gfCNCPoint5[7255] = {X 11.7883, Y 22.2776, Z -7.1667, A 0.000, B 0.000, C 0.000 }
gfCNCPoint5[7256] = {X 14.1139, Y 22.1583, Z -7.1667, A 0.000, B 0.000, C 0.000 }
gfCNCPoint5[7257] = {X 16.4362, Y 21.9881, Z -7.1667, A 0.000, B 0.000, C 0.000 }
gfCNCPoint5[7258] = {X 17.0855, Y 21.9056, Z -7.1667, A 0.000, B 0.000, C 0.000 }
gfCNCPoint5[7259] = {X 17.7182, Y 21.7381, Z -7.1667, A 0.000, B 0.000, C 0.000 }
gfCNCPoint5[7260] = {X 17.7565, Y 21.2348, Z -7.1667, A 0.000, B 0.000, C 0.000 }
gfCNCPoint5[7261] = {X 17.6002, Y 20.7548, Z -7.1667, A 0.000, B 0.000, C 0.000 }
gfCNCPoint5[7262] = {X 17.2730, Y 20.3705, Z -7.1667, A 0.000, B 0.000, C 0.000 }
gfCNCPoint5[7263] = {X 16.3395, Y 19.8212, Z -7.1667, A 0.000, B 0.000, C 0.000 }
gfCNCPoint5[7264] = {X 15.3164, Y 19.4659, Z -7.1667, A 0.000, B 0.000, C 0.000 }
gfCNCPoint5[7265] = {X 13.9815, Y 19.2481, Z -7.1667, A 0.000, B 0.000, C 0.000 }
gfCNCPoint5[7266] = {X 12.6299, Y 19.1939, Z -7.1667, A 0.000, B 0.000, C 0.000 }
gfCNCPoint5[7267] = {X 11.2818, Y 19.3044, Z -7.1667, A 0.000, B 0.000, C 0.000 }
gfCNCPoint5[7268] = {X 10.5939, Y 19.4125, Z -7.1667, A 0.000, B 0.000, C 0.000 }
gfCNCPoint5[7269] = {X 9.2120, Y 19.7717, Z -7.1667, A 0.000, B 0.000, C 0.000 }
gfCNCPoint5[7270] = {X 7.9080, Y 20.3531, Z -7.1667, A 0.000, B 0.000, C 0.000 }
gfCNCPoint5[7271] = {X 7.7436, Y 21.1766, Z -7.1667, A 0.000, B 0.000, C 0.000 }
gfCNCPoint5[7272] = {X 7.4229, Y 21.9527, Z -7.1667, A 0.000, B 0.000, C 0.000 }
gfCNCPoint5[7273] = {X 6.9582, Y 22.6522, Z -7.1667, A 0.000, B 0.000, C 0.000 }
gfCNCPoint5[7274] = {X 9.0864, Y 22.4225, Z -7.1667, A 0.000, B 0.000, C 0.000 }
gfCNCPoint5[7275] = {X 11.2233, Y 22.2989, Z -7.1667, A 0.000, B 0.000, C 0.000 }
gfCNCPoint5[7276] = {X 11.5058, Y 22.2886, Z -7.1667, A 0.000, B 0.000, C 0.000 }
gfCNCPoint5[7277] = {X 11.7883, Y 22.2776, Z -7.1667, A 0.000, B 0.000, C 0.000 }
gfCNCPoint5[7278] = {X 15.7558, Y 21.7688, Z -7.1667, A 0.000, B 0.000, C 0.000 }
gfCNCPoint5[7279] = {X 7.7960, Y 22.1697, Z -7.1667, A 0.000, B 0.000, C 0.000 }
gfCNCPoint5[7280] = {X 11.7916, Y 22.3576, Z -7.1667, A 0.000, B 0.000, C 0.000 }
gfCNCPoint5[7281] = {X 14.1184, Y 22.2382, Z -7.1667, A 0.000, B 0.000, C 0.000 }
gfCNCPoint5[7282] = {X 16.4420, Y 22.0679, Z -7.1667, A 0.000, B 0.000, C 0.000 }
gfCNCPoint5[7283] = {X 17.1218, Y 21.9800, Z -7.1667, A 0.000, B 0.000, C 0.000 }
gfCNCPoint5[7284] = {X 17.7833, Y 21.8004, Z -7.1667, A 0.000, B 0.000, C 0.000 }
gfCNCPoint5[7285] = {X 17.8390, Y 21.2530, Z -7.1667, A 0.000, B 0.000, C 0.000 }
gfCNCPoint5[7286] = {X 17.6764, Y 20.7273, Z -7.1667, A 0.000, B 0.000, C 0.000 }
gfCNCPoint5[7287] = {X 17.3214, Y 20.3068, Z -7.1667, A 0.000, B 0.000, C 0.000 }
gfCNCPoint5[7288] = {X 16.3736, Y 19.7488, Z -7.1667, A 0.000, B 0.000, C 0.000 }
gfCNCPoint5[7289] = {X 15.3346, Y 19.3880, Z -7.1667, A 0.000, B 0.000, C 0.000 }
gfCNCPoint5[7290] = {X 13.9897, Y 19.1685, Z -7.1667, A 0.000, B 0.000, C 0.000 }
gfCNCPoint5[7291] = {X 12.6281, Y 19.1140, Z -7.1667, A 0.000, B 0.000, C 0.000 }
gfCNCPoint5[7292] = {X 11.2699, Y 19.2253, Z -7.1667, A 0.000, B 0.000, C 0.000 }
gfCNCPoint5[7293] = {X 10.5808, Y 19.3336, Z -7.1667, A 0.000, B 0.000, C 0.000 }
gfCNCPoint5[7294] = {X 9.6302, Y 19.5537, Z -7.1667, A 0.000, B 0.000, C 0.000 }
gfCNCPoint5[7295] = {X 8.7101, Y 19.8784, Z -7.1667, A 0.000, B 0.000, C 0.000 }
gfCNCPoint5[7296] = {X 7.8318, Y 20.3037, Z -7.1667, A 0.000, B 0.000, C 0.000 }
gfCNCPoint5[7297] = {X 7.8284, Y 20.3451, Z -7.1667, A 0.000, B 0.000, C 0.000 }
gfCNCPoint5[7298] = {X 7.6463, Y 21.2196, Z -7.1667, A 0.000, B 0.000, C 0.000 }
gfCNCPoint5[7299] = {X 7.2851, Y 22.0366, Z -7.1667, A 0.000, B 0.000, C 0.000 }
gfCNCPoint5[7300] = {X 6.7608, Y 22.7597, Z -7.1667, A 0.000, B 0.000, C 0.000 }
gfCNCPoint5[7301] = {X 8.9884, Y 22.5110, Z -7.1667, A 0.000, B 0.000, C 0.000 }
gfCNCPoint5[7302] = {X 11.2260, Y 22.3789, Z -7.1667, A 0.000, B 0.000, C 0.000 }
gfCNCPoint5[7303] = {X 11.5088, Y 22.3686, Z -7.1667, A 0.000, B 0.000, C 0.000 }
gfCNCPoint5[7304] = {X 11.7916, Y 22.3576, Z -7.1667, A 0.000, B 0.000, C 0.000 }
gfCNCPoint5[7305] = {X 15.7591, Y 21.8487, Z -7.1667, A 0.000, B 0.000, C 0.000 }
gfCNCPoint5[7306] = {X 7.7992, Y 22.2496, Z -7.1667, A 0.000, B 0.000, C 0.000 }
gfCNCPoint5[7307] = {X 11.7948, Y 22.4375, Z -7.1667, A 0.000, B 0.000, C 0.000 }
gfCNCPoint5[7308] = {X 14.1229, Y 22.3181, Z -7.1667, A 0.000, B 0.000, C 0.000 }
gfCNCPoint5[7309] = {X 16.4478, Y 22.1477, Z -7.1667, A 0.000, B 0.000, C 0.000 }
gfCNCPoint5[7310] = {X 17.1574, Y 22.0544, Z -7.1667, A 0.000, B 0.000, C 0.000 }
gfCNCPoint5[7311] = {X 17.8470, Y 21.8628, Z -7.1667, A 0.000, B 0.000, C 0.000 }
gfCNCPoint5[7312] = {X 17.9254, Y 21.4214, Z -7.1667, A 0.000, B 0.000, C 0.000 }
gfCNCPoint5[7313] = {X 17.8662, Y 20.9770, Z -7.1667, A 0.000, B 0.000, C 0.000 }
gfCNCPoint5[7314] = {X 17.6750, Y 20.5715, Z -7.1667, A 0.000, B 0.000, C 0.000 }
gfCNCPoint5[7315] = {X 17.3698, Y 20.2431, Z -7.1667, A 0.000, B 0.000, C 0.000 }
gfCNCPoint5[7316] = {X 16.4076, Y 19.6764, Z -7.1667, A 0.000, B 0.000, C 0.000 }
gfCNCPoint5[7317] = {X 15.3528, Y 19.3101, Z -7.1667, A 0.000, B 0.000, C 0.000 }
gfCNCPoint5[7318] = {X 13.9979, Y 19.0889, Z -7.1667, A 0.000, B 0.000, C 0.000 }
gfCNCPoint5[7319] = {X 12.6262, Y 19.0340, Z -7.1667, A 0.000, B 0.000, C 0.000 }
gfCNCPoint5[7320] = {X 11.2580, Y 19.1461, Z -7.1667, A 0.000, B 0.000, C 0.000 }
gfCNCPoint5[7321] = {X 10.5678, Y 19.2546, Z -7.1667, A 0.000, B 0.000, C 0.000 }
gfCNCPoint5[7322] = {X 9.5945, Y 19.4808, Z -7.1667, A 0.000, B 0.000, C 0.000 }
gfCNCPoint5[7323] = {X 8.6531, Y 19.8156, Z -7.1667, A 0.000, B 0.000, C 0.000 }
gfCNCPoint5[7324] = {X 7.7555, Y 20.2547, Z -7.1667, A 0.000, B 0.000, C 0.000 }
gfCNCPoint5[7325] = {X 7.7492, Y 20.3327, Z -7.1667, A 0.000, B 0.000, C 0.000 }
gfCNCPoint5[7326] = {X 7.5473, Y 21.2643, Z -7.1667, A 0.000, B 0.000, C 0.000 }
gfCNCPoint5[7327] = {X 7.1386, Y 22.1254, Z -7.1667, A 0.000, B 0.000, C 0.000 }
gfCNCPoint5[7328] = {X 6.5446, Y 22.8710, Z -7.1667, A 0.000, B 0.000, C 0.000 }
gfCNCPoint5[7329] = {X 8.8810, Y 22.6006, Z -7.1667, A 0.000, B 0.000, C 0.000 }
gfCNCPoint5[7330] = {X 11.2288, Y 22.4588, Z -7.1667, A 0.000, B 0.000, C 0.000 }
gfCNCPoint5[7331] = {X 11.5118, Y 22.4485, Z -7.1667, A 0.000, B 0.000, C 0.000 }
gfCNCPoint5[7332] = {X 11.7948, Y 22.4375, Z -7.1667, A 0.000, B 0.000, C 0.000 }
gfCNCPoint5[7333] = {X 15.7623, Y 21.9287, Z -7.1667, A 0.000, B 0.000, C 0.000 }
gfCNCPoint5[7334] = {X 7.8024, Y 22.3296, Z -7.1667, A 0.000, B 0.000, C 0.000 }
gfCNCPoint5[7335] = {X 11.7980, Y 22.5174, Z -7.1667, A 0.000, B 0.000, C 0.000 }
gfCNCPoint5[7336] = {X 14.1274, Y 22.3980, Z -7.1667, A 0.000, B 0.000, C 0.000 }
gfCNCPoint5[7337] = {X 16.4536, Y 22.2275, Z -7.1667, A 0.000, B 0.000, C 0.000 }
gfCNCPoint5[7338] = {X 17.1925, Y 22.1289, Z -7.1667, A 0.000, B 0.000, C 0.000 }
gfCNCPoint5[7339] = {X 17.9096, Y 21.9253, Z -7.1667, A 0.000, B 0.000, C 0.000 }
gfCNCPoint5[7340] = {X 18.0045, Y 21.4519, Z -7.1667, A 0.000, B 0.000, C 0.000 }
gfCNCPoint5[7341] = {X 17.9481, Y 20.9724, Z -7.1667, A 0.000, B 0.000, C 0.000 }
gfCNCPoint5[7342] = {X 17.7461, Y 20.5338, Z -7.1667, A 0.000, B 0.000, C 0.000 }
gfCNCPoint5[7343] = {X 17.4182, Y 20.1794, Z -7.1667, A 0.000, B 0.000, C 0.000 }
gfCNCPoint5[7344] = {X 16.4416, Y 19.6040, Z -7.1667, A 0.000, B 0.000, C 0.000 }
gfCNCPoint5[7345] = {X 15.3709, Y 19.2322, Z -7.1667, A 0.000, B 0.000, C 0.000 }
gfCNCPoint5[7346] = {X 14.0061, Y 19.0093, Z -7.1667, A 0.000, B 0.000, C 0.000 }
gfCNCPoint5[7347] = {X 12.6243, Y 18.9540, Z -7.1667, A 0.000, B 0.000, C 0.000 }
gfCNCPoint5[7348] = {X 11.2461, Y 19.0670, Z -7.1667, A 0.000, B 0.000, C 0.000 }
gfCNCPoint5[7349] = {X 10.5547, Y 19.1757, Z -7.1667, A 0.000, B 0.000, C 0.000 }
gfCNCPoint5[7350] = {X 9.5588, Y 19.4079, Z -7.1667, A 0.000, B 0.000, C 0.000 }
gfCNCPoint5[7351] = {X 8.5961, Y 19.7528, Z -7.1667, A 0.000, B 0.000, C 0.000 }
gfCNCPoint5[7352] = {X 7.6793, Y 20.2059, Z -7.1667, A 0.000, B 0.000, C 0.000 }
gfCNCPoint5[7353] = {X 7.6695, Y 20.3255, Z -7.1667, A 0.000, B 0.000, C 0.000 }
gfCNCPoint5[7354] = {X 7.5231, Y 21.0760, Z -7.1667, A 0.000, B 0.000, C 0.000 }
gfCNCPoint5[7355] = {X 7.2392, Y 21.7861, Z -7.1667, A 0.000, B 0.000, C 0.000 }
gfCNCPoint5[7356] = {X 6.8279, Y 22.4307, Z -7.1667, A 0.000, B 0.000, C 0.000 }
gfCNCPoint5[7357] = {X 6.3034, Y 22.9872, Z -7.1667, A 0.000, B 0.000, C 0.000 }
gfCNCPoint5[7358] = {X 8.7610, Y 22.6917, Z -7.1667, A 0.000, B 0.000, C 0.000 }
gfCNCPoint5[7359] = {X 11.2315, Y 22.5388, Z -7.1667, A 0.000, B 0.000, C 0.000 }
gfCNCPoint5[7360] = {X 11.5147, Y 22.5285, Z -7.1667, A 0.000, B 0.000, C 0.000 }
gfCNCPoint5[7361] = {X 11.7980, Y 22.5174, Z -7.1667, A 0.000, B 0.000, C 0.000 }
gfCNCPoint5[7362] = {X 15.7655, Y 22.0086, Z -7.1667, A 0.000, B 0.000, C 0.000 }
gfCNCPoint5[7363] = {X 11.7262, Y 22.6004, Z -7.1667, A 0.000, B 0.000, C 0.000 }
gfCNCPoint5[7364] = {X 11.8012, Y 22.5974, Z -7.1667, A 0.000, B 0.000, C 0.000 }
gfCNCPoint5[7365] = {X 14.1319, Y 22.4778, Z -7.1667, A 0.000, B 0.000, C 0.000 }
gfCNCPoint5[7366] = {X 16.4593, Y 22.3073, Z -7.1667, A 0.000, B 0.000, C 0.000 }
gfCNCPoint5[7367] = {X 17.2271, Y 22.2034, Z -7.1667, A 0.000, B 0.000, C 0.000 }
gfCNCPoint5[7368] = {X 17.9713, Y 21.9879, Z -7.1667, A 0.000, B 0.000, C 0.000 }
gfCNCPoint5[7369] = {X 18.0831, Y 21.4827, Z -7.1667, A 0.000, B 0.000, C 0.000 }
gfCNCPoint5[7370] = {X 18.0299, Y 20.9679, Z -7.1667, A 0.000, B 0.000, C 0.000 }
gfCNCPoint5[7371] = {X 17.8171, Y 20.4962, Z -7.1667, A 0.000, B 0.000, C 0.000 }
gfCNCPoint5[7372] = {X 17.4665, Y 20.1156, Z -7.1667, A 0.000, B 0.000, C 0.000 }
gfCNCPoint5[7373] = {X 16.4756, Y 19.5316, Z -7.1667, A 0.000, B 0.000, C 0.000 }
gfCNCPoint5[7374] = {X 15.3891, Y 19.1542, Z -7.1667, A 0.000, B 0.000, C 0.000 }
gfCNCPoint5[7375] = {X 14.0143, Y 18.9297, Z -7.1667, A 0.000, B 0.000, C 0.000 }
gfCNCPoint5[7376] = {X 12.6225, Y 18.8740, Z -7.1667, A 0.000, B 0.000, C 0.000 }
gfCNCPoint5[7377] = {X 11.2342, Y 18.9879, Z -7.1667, A 0.000, B 0.000, C 0.000 }
gfCNCPoint5[7378] = {X 10.5417, Y 19.0968, Z -7.1667, A 0.000, B 0.000, C 0.000 }
gfCNCPoint5[7379] = {X 9.5230, Y 19.3351, Z -7.1667, A 0.000, B 0.000, C 0.000 }
gfCNCPoint5[7380] = {X 8.5390, Y 19.6902, Z -7.1667, A 0.000, B 0.000, C 0.000 }
gfCNCPoint5[7381] = {X 7.6029, Y 20.1573, Z -7.1667, A 0.000, B 0.000, C 0.000 }
gfCNCPoint5[7382] = {X 7.5898, Y 20.3183, Z -7.1667, A 0.000, B 0.000, C 0.000 }
gfCNCPoint5[7383] = {X 7.4462, Y 21.0539, Z -7.1667, A 0.000, B 0.000, C 0.000 }
gfCNCPoint5[7384] = {X 7.1679, Y 21.7499, Z -7.1667, A 0.000, B 0.000, C 0.000 }
gfCNCPoint5[7385] = {X 6.7646, Y 22.3816, Z -7.1667, A 0.000, B 0.000, C 0.000 }
gfCNCPoint5[7386] = {X 6.2506, Y 22.9271, Z -7.1667, A 0.000, B 0.000, C 0.000 }
gfCNCPoint5[7387] = {X 6.2084, Y 22.9636, Z -7.1667, A 0.000, B 0.000, C 0.000 }
gfCNCPoint5[7388] = {X 6.1658, Y 22.9996, Z -7.1667, A 0.000, B 0.000, C 0.000 }
gfCNCPoint5[7389] = {X 6.1510, Y 23.0912, Z -7.1667, A 0.000, B 0.000, C 0.000 }
gfCNCPoint5[7390] = {X 6.2331, Y 23.0787, Z -7.1667, A 0.000, B 0.000, C 0.000 }
gfCNCPoint5[7391] = {X 6.3153, Y 23.0663, Z -7.1667, A 0.000, B 0.000, C 0.000 }
gfCNCPoint5[7392] = {X 8.7682, Y 22.7714, Z -7.1667, A 0.000, B 0.000, C 0.000 }
gfCNCPoint5[7393] = {X 11.2342, Y 22.6187, Z -7.1667, A 0.000, B 0.000, C 0.000 }
gfCNCPoint5[7394] = {X 11.5177, Y 22.6084, Z -7.1667, A 0.000, B 0.000, C 0.000 }
gfCNCPoint5[7395] = {X 11.8012, Y 22.5974, Z -7.1667, A 0.000, B 0.000, C 0.000 }
gfCNCPoint5[7396] = {X 11.7207, Y 20.5990, Z -7.1667, A 0.000, B 0.000, C 0.000 }
gfCNCPoint5[7397] = {X 11.7207, Y 20.5990, Z -4.1667, A 0.000, B 0.000, C 0.000 }
gfCNCPoint5[7398] = {X 11.7207, Y 20.5990, Z 11.0000, A 0.000, B 0.000, C 0.000 }
gfCNCPoint5[7399] = {X 11.7081, Y 37.8758, Z 11.0000, A 0.000, B 0.000, C 0.000 }
gfCNCPoint5[7400] = {X 11.7081, Y 37.8758, Z -3.3333, A 0.000, B 0.000, C 0.000 }
gfCNCPoint5[7401] = {X 12.5103, Y 37.9481, Z -3.5492, A 0.000, B 0.000, C 0.000 }
gfCNCPoint5[7402] = {X 14.1625, Y 37.8336, Z -3.9929, A 0.000, B 0.000, C 0.000 }
gfCNCPoint5[7403] = {X 15.7757, Y 37.4587, Z -4.4367, A 0.000, B 0.000, C 0.000 }
gfCNCPoint5[7404] = {X 16.5083, Y 37.1628, Z -4.6484, A 0.000, B 0.000, C 0.000 }
gfCNCPoint5[7405] = {X 17.3399, Y 36.8270, Z -4.8887, A 0.000, B 0.000, C 0.000 }
gfCNCPoint5[7406] = {X 18.2933, Y 36.3172, Z -5.1784, A 0.000, B 0.000, C 0.000 }
gfCNCPoint5[7407] = {X 19.0345, Y 35.8122, Z -5.4187, A 0.000, B 0.000, C 0.000 }
gfCNCPoint5[7408] = {X 19.0577, Y 35.2981, Z -5.5566, A 0.000, B 0.000, C 0.000 }
gfCNCPoint5[7409] = {X 19.2187, Y 34.6361, Z -5.7392, A 0.000, B 0.000, C 0.000 }
gfCNCPoint5[7410] = {X 19.4342, Y 34.1687, Z -5.8771, A 0.000, B 0.000, C 0.000 }
gfCNCPoint5[7411] = {X 18.2036, Y 34.4169, Z -6.2135, A 0.000, B 0.000, C 0.000 }
gfCNCPoint5[7412] = {X 17.3629, Y 34.5312, Z -6.4408, A 0.000, B 0.000, C 0.000 }
gfCNCPoint5[7413] = {X 16.1106, Y 34.6206, Z -6.7772, A 0.000, B 0.000, C 0.000 }
gfCNCPoint5[7414] = {X 15.3858, Y 34.6743, Z -6.9719, A 0.000, B 0.000, C 0.000 }
gfCNCPoint5[7415] = {X 14.6608, Y 34.7239, Z -7.1667, A 0.000, B 0.000, C 0.000 }
gfCNCPoint5[7416] = {X 12.2606, Y 34.8765, Z -7.1667, A 0.000, B 0.000, C 0.000 }
gfCNCPoint5[7417] = {X 9.8591, Y 35.0062, Z -7.1667, A 0.000, B 0.000, C 0.000 }
gfCNCPoint5[7418] = {X 8.7540, Y 35.0961, Z -7.1667, A 0.000, B 0.000, C 0.000 }
gfCNCPoint5[7419] = {X 7.6661, Y 35.3099, Z -7.1667, A 0.000, B 0.000, C 0.000 }
gfCNCPoint5[7420] = {X 7.6566, Y 35.3714, Z -7.1667, A 0.000, B 0.000, C 0.000 }
gfCNCPoint5[7421] = {X 7.6532, Y 35.4336, Z -7.1667, A 0.000, B 0.000, C 0.000 }
gfCNCPoint5[7422] = {X 7.7538, Y 36.0257, Z -7.1667, A 0.000, B 0.000, C 0.000 }
gfCNCPoint5[7423] = {X 8.0477, Y 36.5493, Z -7.1667, A 0.000, B 0.000, C 0.000 }
gfCNCPoint5[7424] = {X 8.5008, Y 36.9435, Z -7.1667, A 0.000, B 0.000, C 0.000 }
gfCNCPoint5[7425] = {X 9.2728, Y 37.3352, Z -7.1667, A 0.000, B 0.000, C 0.000 }
gfCNCPoint5[7426] = {X 10.0944, Y 37.6075, Z -7.1667, A 0.000, B 0.000, C 0.000 }
gfCNCPoint5[7427] = {X 11.3792, Y 37.8446, Z -7.1667, A 0.000, B 0.000, C 0.000 }
gfCNCPoint5[7428] = {X 12.6835, Y 37.9185, Z -7.1667, A 0.000, B 0.000, C 0.000 }
gfCNCPoint5[7429] = {X 13.9869, Y 37.8281, Z -7.1667, A 0.000, B 0.000, C 0.000 }
gfCNCPoint5[7430] = {X 15.2685, Y 37.5749, Z -7.1667, A 0.000, B 0.000, C 0.000 }
gfCNCPoint5[7431] = {X 16.5083, Y 37.1628, Z -7.1667, A 0.000, B 0.000, C 0.000 }
gfCNCPoint5[7432] = {X 17.8076, Y 36.5552, Z -7.1667, A 0.000, B 0.000, C 0.000 }
gfCNCPoint5[7433] = {X 19.0345, Y 35.8122, Z -7.1667, A 0.000, B 0.000, C 0.000 }
gfCNCPoint5[7434] = {X 19.1546, Y 34.9711, Z -7.1667, A 0.000, B 0.000, C 0.000 }
gfCNCPoint5[7435] = {X 19.4342, Y 34.1687, Z -7.1667, A 0.000, B 0.000, C 0.000 }
gfCNCPoint5[7436] = {X 17.7796, Y 34.4478, Z -7.1667, A 0.000, B 0.000, C 0.000 }
gfCNCPoint5[7437] = {X 16.1106, Y 34.6206, Z -7.1667, A 0.000, B 0.000, C 0.000 }
gfCNCPoint5[7438] = {X 15.3858, Y 34.6733, Z -7.1667, A 0.000, B 0.000, C 0.000 }
gfCNCPoint5[7439] = {X 14.6608, Y 34.7239, Z -7.1667, A 0.000, B 0.000, C 0.000 }
gfCNCPoint5[7440] = {X 18.6546, Y 34.7200, Z -7.1667, A 0.000, B 0.000, C 0.000 }
gfCNCPoint5[7441] = {X 14.6553, Y 34.6441, Z -7.1667, A 0.000, B 0.000, C 0.000 }
gfCNCPoint5[7442] = {X 12.2588, Y 34.7965, Z -7.1667, A 0.000, B 0.000, C 0.000 }
gfCNCPoint5[7443] = {X 9.8610, Y 34.9261, Z -7.1667, A 0.000, B 0.000, C 0.000 }
gfCNCPoint5[7444] = {X 8.7212, Y 35.0199, Z -7.1667, A 0.000, B 0.000, C 0.000 }
gfCNCPoint5[7445] = {X 7.5998, Y 35.2444, Z -7.1667, A 0.000, B 0.000, C 0.000 }
gfCNCPoint5[7446] = {X 7.5801, Y 35.3380, Z -7.1667, A 0.000, B 0.000, C 0.000 }
gfCNCPoint5[7447] = {X 7.5732, Y 35.4334, Z -7.1667, A 0.000, B 0.000, C 0.000 }
gfCNCPoint5[7448] = {X 7.6783, Y 36.0524, Z -7.1667, A 0.000, B 0.000, C 0.000 }
gfCNCPoint5[7449] = {X 7.9857, Y 36.5999, Z -7.1667, A 0.000, B 0.000, C 0.000 }
gfCNCPoint5[7450] = {X 8.4594, Y 37.0119, Z -7.1667, A 0.000, B 0.000, C 0.000 }
gfCNCPoint5[7451] = {X 9.2420, Y 37.4090, Z -7.1667, A 0.000, B 0.000, C 0.000 }
gfCNCPoint5[7452] = {X 10.0750, Y 37.6851, Z -7.1667, A 0.000, B 0.000, C 0.000 }
gfCNCPoint5[7453] = {X 11.3696, Y 37.9240, Z -7.1667, A 0.000, B 0.000, C 0.000 }
gfCNCPoint5[7454] = {X 12.6840, Y 37.9985, Z -7.1667, A 0.000, B 0.000, C 0.000 }
gfCNCPoint5[7455] = {X 13.9974, Y 37.9074, Z -7.1667, A 0.000, B 0.000, C 0.000 }
gfCNCPoint5[7456] = {X 15.2890, Y 37.6522, Z -7.1667, A 0.000, B 0.000, C 0.000 }
gfCNCPoint5[7457] = {X 16.5383, Y 37.2370, Z -7.1667, A 0.000, B 0.000, C 0.000 }
gfCNCPoint5[7458] = {X 17.8631, Y 36.6163, Z -7.1667, A 0.000, B 0.000, C 0.000 }
gfCNCPoint5[7459] = {X 19.1128, Y 35.8556, Z -7.1667, A 0.000, B 0.000, C 0.000 }
gfCNCPoint5[7460] = {X 19.2470, Y 34.9315, Z -7.1667, A 0.000, B 0.000, C 0.000 }
gfCNCPoint5[7461] = {X 19.5767, Y 34.0578, Z -7.1667, A 0.000, B 0.000, C 0.000 }
gfCNCPoint5[7462] = {X 17.8489, Y 34.3575, Z -7.1667, A 0.000, B 0.000, C 0.000 }
gfCNCPoint5[7463] = {X 16.1048, Y 34.5408, Z -7.1667, A 0.000, B 0.000, C 0.000 }
gfCNCPoint5[7464] = {X 15.3801, Y 34.5935, Z -7.1667, A 0.000, B 0.000, C 0.000 }
gfCNCPoint5[7465] = {X 14.6553, Y 34.6441, Z -7.1667, A 0.000, B 0.000, C 0.000 }
gfCNCPoint5[7466] = {X 10.7036, Y 35.2638, Z -7.1667, A 0.000, B 0.000, C 0.000 }
gfCNCPoint5[7467] = {X 18.6491, Y 34.6402, Z -7.1667, A 0.000, B 0.000, C 0.000 }
gfCNCPoint5[7468] = {X 14.6498, Y 34.5643, Z -7.1667, A 0.000, B 0.000, C 0.000 }
gfCNCPoint5[7469] = {X 12.2546, Y 34.7166, Z -7.1667, A 0.000, B 0.000, C 0.000 }
gfCNCPoint5[7470] = {X 9.8581, Y 34.8462, Z -7.1667, A 0.000, B 0.000, C 0.000 }
gfCNCPoint5[7471] = {X 8.6877, Y 34.9439, Z -7.1667, A 0.000, B 0.000, C 0.000 }
gfCNCPoint5[7472] = {X 7.5368, Y 35.1783, Z -7.1667, A 0.000, B 0.000, C 0.000 }
gfCNCPoint5[7473] = {X 7.5044, Y 35.3039, Z -7.1667, A 0.000, B 0.000, C 0.000 }
gfCNCPoint5[7474] = {X 7.4932, Y 35.4331, Z -7.1667, A 0.000, B 0.000, C 0.000 }
gfCNCPoint5[7475] = {X 7.6029, Y 36.0790, Z -7.1667, A 0.000, B 0.000, C 0.000 }
gfCNCPoint5[7476] = {X 7.9236, Y 36.6504, Z -7.1667, A 0.000, B 0.000, C 0.000 }
gfCNCPoint5[7477] = {X 8.4180, Y 37.0804, Z -7.1667, A 0.000, B 0.000, C 0.000 }
gfCNCPoint5[7478] = {X 9.2112, Y 37.4828, Z -7.1667, A 0.000, B 0.000, C 0.000 }
gfCNCPoint5[7479] = {X 10.0555, Y 37.7627, Z -7.1667, A 0.000, B 0.000, C 0.000 }
gfCNCPoint5[7480] = {X 11.3601, Y 38.0034, Z -7.1667, A 0.000, B 0.000, C 0.000 }
gfCNCPoint5[7481] = {X 12.6845, Y 38.0785, Z -7.1667, A 0.000, B 0.000, C 0.000 }
gfCNCPoint5[7482] = {X 14.0079, Y 37.9867, Z -7.1667, A 0.000, B 0.000, C 0.000 }
gfCNCPoint5[7483] = {X 15.3094, Y 37.7296, Z -7.1667, A 0.000, B 0.000, C 0.000 }
gfCNCPoint5[7484] = {X 16.5682, Y 37.3112, Z -7.1667, A 0.000, B 0.000, C 0.000 }
gfCNCPoint5[7485] = {X 17.9188, Y 36.6772, Z -7.1667, A 0.000, B 0.000, C 0.000 }
gfCNCPoint5[7486] = {X 19.1915, Y 35.8986, Z -7.1667, A 0.000, B 0.000, C 0.000 }
gfCNCPoint5[7487] = {X 19.2642, Y 35.2210, Z -7.1667, A 0.000, B 0.000, C 0.000 }
gfCNCPoint5[7488] = {X 19.4446, Y 34.5638, Z -7.1667, A 0.000, B 0.000, C 0.000 }
gfCNCPoint5[7489] = {X 19.7279, Y 33.9441, Z -7.1667, A 0.000, B 0.000, C 0.000 }
gfCNCPoint5[7490] = {X 17.9225, Y 34.2663, Z -7.1667, A 0.000, B 0.000, C 0.000 }
gfCNCPoint5[7491] = {X 16.0990, Y 34.4610, Z -7.1667, A 0.000, B 0.000, C 0.000 }
gfCNCPoint5[7492] = {X 15.3745, Y 34.5137, Z -7.1667, A 0.000, B 0.000, C 0.000 }
gfCNCPoint5[7493] = {X 14.6498, Y 34.5643, Z -7.1667, A 0.000, B 0.000, C 0.000 }
gfCNCPoint5[7494] = {X 10.6981, Y 35.1839, Z -7.1667, A 0.000, B 0.000, C 0.000 }
gfCNCPoint5[7495] = {X 18.6437, Y 34.5604, Z -7.1667, A 0.000, B 0.000, C 0.000 }
gfCNCPoint5[7496] = {X 14.6444, Y 34.4845, Z -7.1667, A 0.000, B 0.000, C 0.000 }
gfCNCPoint5[7497] = {X 12.2504, Y 34.6367, Z -7.1667, A 0.000, B 0.000, C 0.000 }
gfCNCPoint5[7498] = {X 9.8551, Y 34.7662, Z -7.1667, A 0.000, B 0.000, C 0.000 }
gfCNCPoint5[7499] = {X 8.6554, Y 34.8677, Z -7.1667, A 0.000, B 0.000, C 0.000 }
gfCNCPoint5[7500] = {X 7.4764, Y 35.1116, Z -7.1667, A 0.000, B 0.000, C 0.000 }
gfCNCPoint5[7501] = {X 7.4295, Y 35.2692, Z -7.1667, A 0.000, B 0.000, C 0.000 }
gfCNCPoint5[7502] = {X 7.4132, Y 35.4328, Z -7.1667, A 0.000, B 0.000, C 0.000 }
gfCNCPoint5[7503] = {X 7.5275, Y 36.1057, Z -7.1667, A 0.000, B 0.000, C 0.000 }
gfCNCPoint5[7504] = {X 7.8616, Y 36.7009, Z -7.1667, A 0.000, B 0.000, C 0.000 }
gfCNCPoint5[7505] = {X 8.3766, Y 37.1488, Z -7.1667, A 0.000, B 0.000, C 0.000 }
gfCNCPoint5[7506] = {X 9.1804, Y 37.5567, Z -7.1667, A 0.000, B 0.000, C 0.000 }
gfCNCPoint5[7507] = {X 10.0361, Y 37.8403, Z -7.1667, A 0.000, B 0.000, C 0.000 }
gfCNCPoint5[7508] = {X 11.3506, Y 38.0829, Z -7.1667, A 0.000, B 0.000, C 0.000 }
gfCNCPoint5[7509] = {X 12.6850, Y 38.1585, Z -7.1667, A 0.000, B 0.000, C 0.000 }
gfCNCPoint5[7510] = {X 14.0185, Y 38.0660, Z -7.1667, A 0.000, B 0.000, C 0.000 }
gfCNCPoint5[7511] = {X 15.3298, Y 37.8069, Z -7.1667, A 0.000, B 0.000, C 0.000 }
gfCNCPoint5[7512] = {X 16.5982, Y 37.3853, Z -7.1667, A 0.000, B 0.000, C 0.000 }
gfCNCPoint5[7513] = {X 17.9747, Y 36.7379, Z -7.1667, A 0.000, B 0.000, C 0.000 }
gfCNCPoint5[7514] = {X 19.2706, Y 35.9411, Z -7.1667, A 0.000, B 0.000, C 0.000 }
gfCNCPoint5[7515] = {X 19.3492, Y 35.2031, Z -7.1667, A 0.000, B 0.000, C 0.000 }
gfCNCPoint5[7516] = {X 19.5577, Y 34.4908, Z -7.1667, A 0.000, B 0.000, C 0.000 }
gfCNCPoint5[7517] = {X 19.8895, Y 33.8269, Z -7.1667, A 0.000, B 0.000, C 0.000 }
gfCNCPoint5[7518] = {X 18.0016, Y 34.1741, Z -7.1667, A 0.000, B 0.000, C 0.000 }
gfCNCPoint5[7519] = {X 16.0932, Y 34.3812, Z -7.1667, A 0.000, B 0.000, C 0.000 }
gfCNCPoint5[7520] = {X 15.3689, Y 34.4339, Z -7.1667, A 0.000, B 0.000, C 0.000 }
gfCNCPoint5[7521] = {X 14.6444, Y 34.4845, Z -7.1667, A 0.000, B 0.000, C 0.000 }
gfCNCPoint5[7522] = {X 10.6927, Y 35.1041, Z -7.1667, A 0.000, B 0.000, C 0.000 }
gfCNCPoint5[7523] = {X 18.6382, Y 34.4806, Z -7.1667, A 0.000, B 0.000, C 0.000 }
gfCNCPoint5[7524] = {X 14.6389, Y 34.4047, Z -7.1667, A 0.000, B 0.000, C 0.000 }
gfCNCPoint5[7525] = {X 12.2462, Y 34.5568, Z -7.1667, A 0.000, B 0.000, C 0.000 }
gfCNCPoint5[7526] = {X 9.8522, Y 34.6863, Z -7.1667, A 0.000, B 0.000, C 0.000 }
gfCNCPoint5[7527] = {X 8.6243, Y 34.7914, Z -7.1667, A 0.000, B 0.000, C 0.000 }
gfCNCPoint5[7528] = {X 7.4182, Y 35.0445, Z -7.1667, A 0.000, B 0.000, C 0.000 }
gfCNCPoint5[7529] = {X 7.3551, Y 35.2340, Z -7.1667, A 0.000, B 0.000, C 0.000 }
gfCNCPoint5[7530] = {X 7.3332, Y 35.4325, Z -7.1667, A 0.000, B 0.000, C 0.000 }
gfCNCPoint5[7531] = {X 7.3999, Y 35.9619, Z -7.1667, A 0.000, B 0.000, C 0.000 }
gfCNCPoint5[7532] = {X 7.5992, Y 36.4568, Z -7.1667, A 0.000, B 0.000, C 0.000 }
gfCNCPoint5[7533] = {X 7.9179, Y 36.8847, Z -7.1667, A 0.000, B 0.000, C 0.000 }
gfCNCPoint5[7534] = {X 8.3351, Y 37.2173, Z -7.1667, A 0.000, B 0.000, C 0.000 }
gfCNCPoint5[7535] = {X 9.1497, Y 37.6305, Z -7.1667, A 0.000, B 0.000, C 0.000 }
gfCNCPoint5[7536] = {X 10.0167, Y 37.9179, Z -7.1667, A 0.000, B 0.000, C 0.000 }
gfCNCPoint5[7537] = {X 11.3410, Y 38.1623, Z -7.1667, A 0.000, B 0.000, C 0.000 }
gfCNCPoint5[7538] = {X 12.6856, Y 38.2385, Z -7.1667, A 0.000, B 0.000, C 0.000 }
gfCNCPoint5[7539] = {X 14.0290, Y 38.1453, Z -7.1667, A 0.000, B 0.000, C 0.000 }
gfCNCPoint5[7540] = {X 15.3502, Y 37.8843, Z -7.1667, A 0.000, B 0.000, C 0.000 }
gfCNCPoint5[7541] = {X 16.6281, Y 37.4595, Z -7.1667, A 0.000, B 0.000, C 0.000 }
gfCNCPoint5[7542] = {X 18.0309, Y 36.7984, Z -7.1667, A 0.000, B 0.000, C 0.000 }
gfCNCPoint5[7543] = {X 19.3501, Y 35.9832, Z -7.1667, A 0.000, B 0.000, C 0.000 }
gfCNCPoint5[7544] = {X 19.4352, Y 35.1815, Z -7.1667, A 0.000, B 0.000, C 0.000 }
gfCNCPoint5[7545] = {X 19.6763, Y 34.4122, Z -7.1667, A 0.000, B 0.000, C 0.000 }
gfCNCPoint5[7546] = {X 20.0639, Y 33.7053, Z -7.1667, A 0.000, B 0.000, C 0.000 }
gfCNCPoint5[7547] = {X 18.0872, Y 34.0806, Z -7.1667, A 0.000, B 0.000, C 0.000 }
gfCNCPoint5[7548] = {X 16.0874, Y 34.3014, Z -7.1667, A 0.000, B 0.000, C 0.000 }
gfCNCPoint5[7549] = {X 15.3632, Y 34.3541, Z -7.1667, A 0.000, B 0.000, C 0.000 }
gfCNCPoint5[7550] = {X 14.6389, Y 34.4047, Z -7.1667, A 0.000, B 0.000, C 0.000 }
gfCNCPoint5[7551] = {X 10.6872, Y 35.0243, Z -7.1667, A 0.000, B 0.000, C 0.000 }
gfCNCPoint5[7552] = {X 14.7699, Y 36.3202, Z -7.1667, A 0.000, B 0.000, C 0.000 }
gfCNCPoint5[7553] = {X 14.6335, Y 34.3248, Z -7.1667, A 0.000, B 0.000, C 0.000 }
gfCNCPoint5[7554] = {X 12.2420, Y 34.4770, Z -7.1667, A 0.000, B 0.000, C 0.000 }
gfCNCPoint5[7555] = {X 9.8492, Y 34.6063, Z -7.1667, A 0.000, B 0.000, C 0.000 }
gfCNCPoint5[7556] = {X 8.5941, Y 34.7150, Z -7.1667, A 0.000, B 0.000, C 0.000 }
gfCNCPoint5[7557] = {X 7.3618, Y 34.9771, Z -7.1667, A 0.000, B 0.000, C 0.000 }
gfCNCPoint5[7558] = {X 7.2812, Y 35.1984, Z -7.1667, A 0.000, B 0.000, C 0.000 }
gfCNCPoint5[7559] = {X 7.2532, Y 35.4322, Z -7.1667, A 0.000, B 0.000, C 0.000 }
gfCNCPoint5[7560] = {X 7.3225, Y 35.9820, Z -7.1667, A 0.000, B 0.000, C 0.000 }
gfCNCPoint5[7561] = {X 7.5294, Y 36.4960, Z -7.1667, A 0.000, B 0.000, C 0.000 }
gfCNCPoint5[7562] = {X 7.8604, Y 36.9403, Z -7.1667, A 0.000, B 0.000, C 0.000 }
gfCNCPoint5[7563] = {X 8.2937, Y 37.2857, Z -7.1667, A 0.000, B 0.000, C 0.000 }
gfCNCPoint5[7564] = {X 9.1189, Y 37.7044, Z -7.1667, A 0.000, B 0.000, C 0.000 }
gfCNCPoint5[7565] = {X 9.9973, Y 37.9956, Z -7.1667, A 0.000, B 0.000, C 0.000 }
gfCNCPoint5[7566] = {X 11.3315, Y 38.2417, Z -7.1667, A 0.000, B 0.000, C 0.000 }
gfCNCPoint5[7567] = {X 12.6861, Y 38.3185, Z -7.1667, A 0.000, B 0.000, C 0.000 }
gfCNCPoint5[7568] = {X 14.0396, Y 38.2246, Z -7.1667, A 0.000, B 0.000, C 0.000 }
gfCNCPoint5[7569] = {X 15.3706, Y 37.9617, Z -7.1667, A 0.000, B 0.000, C 0.000 }
gfCNCPoint5[7570] = {X 16.6581, Y 37.5337, Z -7.1667, A 0.000, B 0.000, C 0.000 }
gfCNCPoint5[7571] = {X 18.0873, Y 36.8588, Z -7.1667, A 0.000, B 0.000, C 0.000 }
gfCNCPoint5[7572] = {X 19.4300, Y 36.0248, Z -7.1667, A 0.000, B 0.000, C 0.000 }
gfCNCPoint5[7573] = {X 19.5226, Y 35.1553, Z -7.1667, A 0.000, B 0.000, C 0.000 }
gfCNCPoint5[7574] = {X 19.8019, Y 34.3266, Z -7.1667, A 0.000, B 0.000, C 0.000 }
gfCNCPoint5[7575] = {X 20.2547, Y 33.5784, Z -7.1667, A 0.000, B 0.000, C 0.000 }
gfCNCPoint5[7576] = {X 18.1813, Y 33.9853, Z -7.1667, A 0.000, B 0.000, C 0.000 }
gfCNCPoint5[7577] = {X 16.0816, Y 34.2216, Z -7.1667, A 0.000, B 0.000, C 0.000 }
gfCNCPoint5[7578] = {X 15.3576, Y 34.2743, Z -7.1667, A 0.000, B 0.000, C 0.000 }
gfCNCPoint5[7579] = {X 14.6335, Y 34.3248, Z -7.1667, A 0.000, B 0.000, C 0.000 }
gfCNCPoint5[7580] = {X 14.7699, Y 36.3202, Z -7.1667, A 0.000, B 0.000, C 0.000 }
gfCNCPoint5[7581] = {X 14.7699, Y 36.3202, Z -4.1667, A 0.000, B 0.000, C 0.000 }
gfCNCPoint5[7582] = {X 14.7699, Y 36.3202, Z 11.0000, A 0.000, B 0.000, C 0.000 }
gfCNCPoint5[7583] = {X 165.6772, Y 73.8165, Z 11.0000, A 0.000, B 0.000, C 0.000 }
gfCNCPoint5[7584] = {X 165.6772, Y 73.8165, Z -3.3333, A 0.000, B 0.000, C 0.000 }
gfCNCPoint5[7585] = {X 161.3996, Y 78.5670, Z -5.0462, A 0.000, B 0.000, C 0.000 }
gfCNCPoint5[7586] = {X 169.3132, Y 78.5670, Z -7.1667, A 0.000, B 0.000, C 0.000 }
gfCNCPoint5[7587] = {X 169.3132, Y 76.1670, Z -7.1667, A 0.000, B 0.000, C 0.000 }
gfCNCPoint5[7588] = {X 171.8361, Y 76.1670, Z -7.1667, A 0.000, B 0.000, C 0.000 }
gfCNCPoint5[7589] = {X 169.3147, Y 73.3634, Z -7.1667, A 0.000, B 0.000, C 0.000 }
gfCNCPoint5[7590] = {X 166.7903, Y 76.1670, Z -7.1667, A 0.000, B 0.000, C 0.000 }
gfCNCPoint5[7591] = {X 169.3132, Y 76.1670, Z -7.1667, A 0.000, B 0.000, C 0.000 }
gfCNCPoint5[7592] = {X 169.3132, Y 78.5670, Z -7.1667, A 0.000, B 0.000, C 0.000 }
gfCNCPoint5[7593] = {X 177.2224, Y 78.5670, Z -7.1667, A 0.000, B 0.000, C 0.000 }
gfCNCPoint5[7594] = {X 169.3158, Y 69.7756, Z -7.1667, A 0.000, B 0.000, C 0.000 }
gfCNCPoint5[7595] = {X 161.3996, Y 78.5670, Z -7.1667, A 0.000, B 0.000, C 0.000 }
gfCNCPoint5[7596] = {X 169.3132, Y 78.5670, Z -7.1667, A 0.000, B 0.000, C 0.000 }
gfCNCPoint5[7597] = {X 169.3132, Y 74.6470, Z -7.1667, A 0.000, B 0.000, C 0.000 }
gfCNCPoint5[7598] = {X 169.3132, Y 78.6470, Z -7.1667, A 0.000, B 0.000, C 0.000 }
gfCNCPoint5[7599] = {X 177.4019, Y 78.6470, Z -7.1667, A 0.000, B 0.000, C 0.000 }
gfCNCPoint5[7600] = {X 169.3159, Y 69.6560, Z -7.1667, A 0.000, B 0.000, C 0.000 }
gfCNCPoint5[7601] = {X 161.2199, Y 78.6470, Z -7.1667, A 0.000, B 0.000, C 0.000 }
gfCNCPoint5[7602] = {X 169.3132, Y 78.6470, Z -7.1667, A 0.000, B 0.000, C 0.000 }
gfCNCPoint5[7603] = {X 169.3132, Y 74.6470, Z -7.1667, A 0.000, B 0.000, C 0.000 }
gfCNCPoint5[7604] = {X 169.3132, Y 74.7270, Z -7.1667, A 0.000, B 0.000, C 0.000 }
gfCNCPoint5[7605] = {X 169.3132, Y 78.7270, Z -7.1667, A 0.000, B 0.000, C 0.000 }
gfCNCPoint5[7606] = {X 177.5814, Y 78.7270, Z -7.1667, A 0.000, B 0.000, C 0.000 }
gfCNCPoint5[7607] = {X 169.3159, Y 69.5364, Z -7.1667, A 0.000, B 0.000, C 0.000 }
gfCNCPoint5[7608] = {X 161.0403, Y 78.7270, Z -7.1667, A 0.000, B 0.000, C 0.000 }
gfCNCPoint5[7609] = {X 169.3132, Y 78.7270, Z -7.1667, A 0.000, B 0.000, C 0.000 }
gfCNCPoint5[7610] = {X 169.3132, Y 74.7270, Z -7.1667, A 0.000, B 0.000, C 0.000 }
gfCNCPoint5[7611] = {X 169.3132, Y 74.8070, Z -7.1667, A 0.000, B 0.000, C 0.000 }
gfCNCPoint5[7612] = {X 169.3132, Y 78.8070, Z -7.1667, A 0.000, B 0.000, C 0.000 }
gfCNCPoint5[7613] = {X 177.7610, Y 78.8070, Z -7.1667, A 0.000, B 0.000, C 0.000 }
gfCNCPoint5[7614] = {X 169.3159, Y 69.4168, Z -7.1667, A 0.000, B 0.000, C 0.000 }
gfCNCPoint5[7615] = {X 160.8606, Y 78.8070, Z -7.1667, A 0.000, B 0.000, C 0.000 }
gfCNCPoint5[7616] = {X 169.3132, Y 78.8070, Z -7.1667, A 0.000, B 0.000, C 0.000 }
gfCNCPoint5[7617] = {X 169.3132, Y 74.8070, Z -7.1667, A 0.000, B 0.000, C 0.000 }
gfCNCPoint5[7618] = {X 169.3132, Y 74.8870, Z -7.1667, A 0.000, B 0.000, C 0.000 }
gfCNCPoint5[7619] = {X 169.3132, Y 78.8870, Z -7.1667, A 0.000, B 0.000, C 0.000 }
gfCNCPoint5[7620] = {X 177.9405, Y 78.8870, Z -7.1667, A 0.000, B 0.000, C 0.000 }
gfCNCPoint5[7621] = {X 169.3160, Y 69.2972, Z -7.1667, A 0.000, B 0.000, C 0.000 }
gfCNCPoint5[7622] = {X 160.6809, Y 78.8870, Z -7.1667, A 0.000, B 0.000, C 0.000 }
gfCNCPoint5[7623] = {X 169.3132, Y 78.8870, Z -7.1667, A 0.000, B 0.000, C 0.000 }
gfCNCPoint5[7624] = {X 169.3132, Y 74.8870, Z -7.1667, A 0.000, B 0.000, C 0.000 }
gfCNCPoint5[7625] = {X 169.3132, Y 74.9670, Z -7.1667, A 0.000, B 0.000, C 0.000 }
gfCNCPoint5[7626] = {X 169.3132, Y 78.9670, Z -7.1667, A 0.000, B 0.000, C 0.000 }
gfCNCPoint5[7627] = {X 178.1201, Y 78.9670, Z -7.1667, A 0.000, B 0.000, C 0.000 }
gfCNCPoint5[7628] = {X 169.3160, Y 69.1776, Z -7.1667, A 0.000, B 0.000, C 0.000 }
gfCNCPoint5[7629] = {X 160.5012, Y 78.9670, Z -7.1667, A 0.000, B 0.000, C 0.000 }
gfCNCPoint5[7630] = {X 169.3132, Y 78.9670, Z -7.1667, A 0.000, B 0.000, C 0.000 }
gfCNCPoint5[7631] = {X 169.3132, Y 74.9670, Z -7.1667, A 0.000, B 0.000, C 0.000 }
gfCNCPoint5[7632] = {X 169.3132, Y 74.9670, Z -4.1667, A 0.000, B 0.000, C 0.000 }
gfCNCPoint5[7633] = {X 169.3132, Y 74.9670, Z 11.0000, A 0.000, B 0.000, C 0.000 }
gfCNCPoint5[7634] = {X 186.2261, Y 37.9115, Z 11.0000, A 0.000, B 0.000, C 0.000 }
gfCNCPoint5[7635] = {X 186.2261, Y 37.9115, Z -3.3333, A 0.000, B 0.000, C 0.000 }
gfCNCPoint5[7636] = {X 187.6031, Y 37.8294, Z -3.7030, A 0.000, B 0.000, C 0.000 }
gfCNCPoint5[7637] = {X 189.4361, Y 37.3783, Z -4.2088, A 0.000, B 0.000, C 0.000 }
gfCNCPoint5[7638] = {X 191.0017, Y 36.7012, Z -4.6658, A 0.000, B 0.000, C 0.000 }
gfCNCPoint5[7639] = {X 191.6877, Y 36.3251, Z -4.8755, A 0.000, B 0.000, C 0.000 }
gfCNCPoint5[7640] = {X 192.4467, Y 35.8115, Z -5.1210, A 0.000, B 0.000, C 0.000 }
gfCNCPoint5[7641] = {X 192.4700, Y 35.2974, Z -5.2589, A 0.000, B 0.000, C 0.000 }
gfCNCPoint5[7642] = {X 192.6310, Y 34.6359, Z -5.4413, A 0.000, B 0.000, C 0.000 }
gfCNCPoint5[7643] = {X 192.8465, Y 34.1685, Z -5.5792, A 0.000, B 0.000, C 0.000 }
gfCNCPoint5[7644] = {X 192.7389, Y 34.1935, Z -5.6089, A 0.000, B 0.000, C 0.000 }
gfCNCPoint5[7645] = {X 191.4065, Y 34.4439, Z -5.9721, A 0.000, B 0.000, C 0.000 }
gfCNCPoint5[7646] = {X 190.5829, Y 34.5499, Z -6.1946, A 0.000, B 0.000, C 0.000 }
gfCNCPoint5[7647] = {X 189.2271, Y 34.6452, Z -6.5588, A 0.000, B 0.000, C 0.000 }
gfCNCPoint5[7648] = {X 186.9628, Y 34.7842, Z -7.1667, A 0.000, B 0.000, C 0.000 }
gfCNCPoint5[7649] = {X 182.5915, Y 35.0526, Z -7.1667, A 0.000, B 0.000, C 0.000 }
gfCNCPoint5[7650] = {X 181.8257, Y 35.1406, Z -7.1667, A 0.000, B 0.000, C 0.000 }
gfCNCPoint5[7651] = {X 181.0736, Y 35.3090, Z -7.1667, A 0.000, B 0.000, C 0.000 }
gfCNCPoint5[7652] = {X 181.0656, Y 35.3828, Z -7.1667, A 0.000, B 0.000, C 0.000 }
gfCNCPoint5[7653] = {X 181.0658, Y 35.4571, Z -7.1667, A 0.000, B 0.000, C 0.000 }
gfCNCPoint5[7654] = {X 181.1583, Y 35.9997, Z -7.1667, A 0.000, B 0.000, C 0.000 }
gfCNCPoint5[7655] = {X 181.4151, Y 36.4865, Z -7.1667, A 0.000, B 0.000, C 0.000 }
gfCNCPoint5[7656] = {X 181.8108, Y 36.8691, Z -7.1667, A 0.000, B 0.000, C 0.000 }
gfCNCPoint5[7657] = {X 182.4283, Y 37.2221, Z -7.1667, A 0.000, B 0.000, C 0.000 }
gfCNCPoint5[7658] = {X 183.0886, Y 37.4865, Z -7.1667, A 0.000, B 0.000, C 0.000 }
gfCNCPoint5[7659] = {X 184.4988, Y 37.8010, Z -7.1667, A 0.000, B 0.000, C 0.000 }
gfCNCPoint5[7660] = {X 185.9391, Y 37.9163, Z -7.1667, A 0.000, B 0.000, C 0.000 }
gfCNCPoint5[7661] = {X 187.3814, Y 37.8304, Z -7.1667, A 0.000, B 0.000, C 0.000 }
gfCNCPoint5[7662] = {X 188.7977, Y 37.5447, Z -7.1667, A 0.000, B 0.000, C 0.000 }
gfCNCPoint5[7663] = {X 190.1606, Y 37.0650, Z -7.1667, A 0.000, B 0.000, C 0.000 }
gfCNCPoint5[7664] = {X 191.3329, Y 36.4917, Z -7.1667, A 0.000, B 0.000, C 0.000 }
gfCNCPoint5[7665] = {X 192.4467, Y 35.8115, Z -7.1667, A 0.000, B 0.000, C 0.000 }
gfCNCPoint5[7666] = {X 192.5669, Y 34.9706, Z -7.1667, A 0.000, B 0.000, C 0.000 }
gfCNCPoint5[7667] = {X 192.8465, Y 34.1685, Z -7.1667, A 0.000, B 0.000, C 0.000 }
gfCNCPoint5[7668] = {X 192.7389, Y 34.1935, Z -7.1667, A 0.000, B 0.000, C 0.000 }
gfCNCPoint5[7669] = {X 190.9895, Y 34.4702, Z -7.1667, A 0.000, B 0.000, C 0.000 }
gfCNCPoint5[7670] = {X 189.2271, Y 34.6452, Z -7.1667, A 0.000, B 0.000, C 0.000 }
gfCNCPoint5[7671] = {X 186.9628, Y 34.7842, Z -7.1667, A 0.000, B 0.000, C 0.000 }
gfCNCPoint5[7672] = {X 190.9565, Y 34.8081, Z -7.1667, A 0.000, B 0.000, C 0.000 }
gfCNCPoint5[7673] = {X 186.9579, Y 34.7044, Z -7.1667, A 0.000, B 0.000, C 0.000 }
gfCNCPoint5[7674] = {X 182.5866, Y 34.9728, Z -7.1667, A 0.000, B 0.000, C 0.000 }
gfCNCPoint5[7675] = {X 181.7881, Y 35.0658, Z -7.1667, A 0.000, B 0.000, C 0.000 }
gfCNCPoint5[7676] = {X 181.0046, Y 35.2455, Z -7.1667, A 0.000, B 0.000, C 0.000 }
gfCNCPoint5[7677] = {X 180.9880, Y 35.3486, Z -7.1667, A 0.000, B 0.000, C 0.000 }
gfCNCPoint5[7678] = {X 180.9857, Y 35.4529, Z -7.1667, A 0.000, B 0.000, C 0.000 }
gfCNCPoint5[7679] = {X 181.0816, Y 36.0225, Z -7.1667, A 0.000, B 0.000, C 0.000 }
gfCNCPoint5[7680] = {X 181.3505, Y 36.5336, Z -7.1667, A 0.000, B 0.000, C 0.000 }
gfCNCPoint5[7681] = {X 181.7657, Y 36.9352, Z -7.1667, A 0.000, B 0.000, C 0.000 }
gfCNCPoint5[7682] = {X 182.3935, Y 37.2941, Z -7.1667, A 0.000, B 0.000, C 0.000 }
gfCNCPoint5[7683] = {X 183.0649, Y 37.5629, Z -7.1667, A 0.000, B 0.000, C 0.000 }
gfCNCPoint5[7684] = {X 184.4862, Y 37.8800, Z -7.1667, A 0.000, B 0.000, C 0.000 }
gfCNCPoint5[7685] = {X 185.9377, Y 37.9963, Z -7.1667, A 0.000, B 0.000, C 0.000 }
gfCNCPoint5[7686] = {X 187.3913, Y 37.9097, Z -7.1667, A 0.000, B 0.000, C 0.000 }
gfCNCPoint5[7687] = {X 188.8188, Y 37.6219, Z -7.1667, A 0.000, B 0.000, C 0.000 }
gfCNCPoint5[7688] = {X 190.1924, Y 37.1384, Z -7.1667, A 0.000, B 0.000, C 0.000 }
gfCNCPoint5[7689] = {X 191.3891, Y 36.5521, Z -7.1667, A 0.000, B 0.000, C 0.000 }
gfCNCPoint5[7690] = {X 192.5250, Y 35.8551, Z -7.1667, A 0.000, B 0.000, C 0.000 }
gfCNCPoint5[7691] = {X 192.6601, Y 34.9279, Z -7.1667, A 0.000, B 0.000, C 0.000 }
gfCNCPoint5[7692] = {X 192.9920, Y 34.0518, Z -7.1667, A 0.000, B 0.000, C 0.000 }
gfCNCPoint5[7693] = {X 192.7315, Y 34.1135, Z -7.1667, A 0.000, B 0.000, C 0.000 }
gfCNCPoint5[7694] = {X 190.9841, Y 34.3902, Z -7.1667, A 0.000, B 0.000, C 0.000 }
gfCNCPoint5[7695] = {X 189.2236, Y 34.5653, Z -7.1667, A 0.000, B 0.000, C 0.000 }
gfCNCPoint5[7696] = {X 186.9579, Y 34.7044, Z -7.1667, A 0.000, B 0.000, C 0.000 }
gfCNCPoint5[7697] = {X 183.0019, Y 35.2966, Z -7.1667, A 0.000, B 0.000, C 0.000 }
gfCNCPoint5[7698] = {X 190.9516, Y 34.7283, Z -7.1667, A 0.000, B 0.000, C 0.000 }
gfCNCPoint5[7699] = {X 186.9529, Y 34.6245, Z -7.1667, A 0.000, B 0.000, C 0.000 }
gfCNCPoint5[7700] = {X 182.5817, Y 34.8929, Z -7.1667, A 0.000, B 0.000, C 0.000 }
gfCNCPoint5[7701] = {X 181.7521, Y 34.9909, Z -7.1667, A 0.000, B 0.000, C 0.000 }
gfCNCPoint5[7702] = {X 180.9387, Y 35.1813, Z -7.1667, A 0.000, B 0.000, C 0.000 }
gfCNCPoint5[7703] = {X 180.9109, Y 35.3168, Z -7.1667, A 0.000, B 0.000, C 0.000 }
gfCNCPoint5[7704] = {X 180.9057, Y 35.4551, Z -7.1667, A 0.000, B 0.000, C 0.000 }
gfCNCPoint5[7705] = {X 181.0062, Y 36.0493, Z -7.1667, A 0.000, B 0.000, C 0.000 }
gfCNCPoint5[7706] = {X 181.2871, Y 36.5825, Z -7.1667, A 0.000, B 0.000, C 0.000 }
gfCNCPoint5[7707] = {X 181.7205, Y 37.0013, Z -7.1667, A 0.000, B 0.000, C 0.000 }
gfCNCPoint5[7708] = {X 182.3587, Y 37.3662, Z -7.1667, A 0.000, B 0.000, C 0.000 }
gfCNCPoint5[7709] = {X 183.0412, Y 37.6394, Z -7.1667, A 0.000, B 0.000, C 0.000 }
gfCNCPoint5[7710] = {X 184.4735, Y 37.9590, Z -7.1667, A 0.000, B 0.000, C 0.000 }
gfCNCPoint5[7711] = {X 185.9363, Y 38.0763, Z -7.1667, A 0.000, B 0.000, C 0.000 }
gfCNCPoint5[7712] = {X 187.4013, Y 37.9891, Z -7.1667, A 0.000, B 0.000, C 0.000 }
gfCNCPoint5[7713] = {X 188.8399, Y 37.6991, Z -7.1667, A 0.000, B 0.000, C 0.000 }
gfCNCPoint5[7714] = {X 190.2241, Y 37.2119, Z -7.1667, A 0.000, B 0.000, C 0.000 }
gfCNCPoint5[7715] = {X 191.4455, Y 36.6123, Z -7.1667, A 0.000, B 0.000, C 0.000 }
gfCNCPoint5[7716] = {X 192.6036, Y 35.8982, Z -7.1667, A 0.000, B 0.000, C 0.000 }
gfCNCPoint5[7717] = {X 192.6772, Y 35.2166, Z -7.1667, A 0.000, B 0.000, C 0.000 }
gfCNCPoint5[7718] = {X 192.8597, Y 34.5557, Z -7.1667, A 0.000, B 0.000, C 0.000 }
gfCNCPoint5[7719] = {X 193.1463, Y 33.9330, Z -7.1667, A 0.000, B 0.000, C 0.000 }
gfCNCPoint5[7720] = {X 192.7149, Y 34.0352, Z -7.1667, A 0.000, B 0.000, C 0.000 }
gfCNCPoint5[7721] = {X 190.9731, Y 34.3110, Z -7.1667, A 0.000, B 0.000, C 0.000 }
gfCNCPoint5[7722] = {X 189.2183, Y 34.4854, Z -7.1667, A 0.000, B 0.000, C 0.000 }
gfCNCPoint5[7723] = {X 186.9529, Y 34.6245, Z -7.1667, A 0.000, B 0.000, C 0.000 }
gfCNCPoint5[7724] = {X 182.9970, Y 35.2167, Z -7.1667, A 0.000, B 0.000, C 0.000 }
gfCNCPoint5[7725] = {X 190.9467, Y 34.6484, Z -7.1667, A 0.000, B 0.000, C 0.000 }
gfCNCPoint5[7726] = {X 186.9480, Y 34.5447, Z -7.1667, A 0.000, B 0.000, C 0.000 }
gfCNCPoint5[7727] = {X 182.5768, Y 34.8131, Z -7.1667, A 0.000, B 0.000, C 0.000 }
gfCNCPoint5[7728] = {X 181.7173, Y 34.9158, Z -7.1667, A 0.000, B 0.000, C 0.000 }
gfCNCPoint5[7729] = {X 180.8754, Y 35.1167, Z -7.1667, A 0.000, B 0.000, C 0.000 }
gfCNCPoint5[7730] = {X 180.8345, Y 35.2846, Z -7.1667, A 0.000, B 0.000, C 0.000 }
gfCNCPoint5[7731] = {X 180.8257, Y 35.4572, Z -7.1667, A 0.000, B 0.000, C 0.000 }
gfCNCPoint5[7732] = {X 180.9308, Y 36.0761, Z -7.1667, A 0.000, B 0.000, C 0.000 }
gfCNCPoint5[7733] = {X 181.2238, Y 36.6313, Z -7.1667, A 0.000, B 0.000, C 0.000 }
gfCNCPoint5[7734] = {X 181.6754, Y 37.0673, Z -7.1667, A 0.000, B 0.000, C 0.000 }
gfCNCPoint5[7735] = {X 182.3240, Y 37.4382, Z -7.1667, A 0.000, B 0.000, C 0.000 }
gfCNCPoint5[7736] = {X 183.0175, Y 37.7158, Z -7.1667, A 0.000, B 0.000, C 0.000 }
gfCNCPoint5[7737] = {X 184.4609, Y 38.0380, Z -7.1667, A 0.000, B 0.000, C 0.000 }
gfCNCPoint5[7738] = {X 185.9350, Y 38.1563, Z -7.1667, A 0.000, B 0.000, C 0.000 }
gfCNCPoint5[7739] = {X 187.4112, Y 38.0685, Z -7.1667, A 0.000, B 0.000, C 0.000 }
gfCNCPoint5[7740] = {X 188.8609, Y 37.7763, Z -7.1667, A 0.000, B 0.000, C 0.000 }
gfCNCPoint5[7741] = {X 190.2559, Y 37.2853, Z -7.1667, A 0.000, B 0.000, C 0.000 }
gfCNCPoint5[7742] = {X 191.5022, Y 36.6724, Z -7.1667, A 0.000, B 0.000, C 0.000 }
gfCNCPoint5[7743] = {X 192.6827, Y 35.9409, Z -7.1667, A 0.000, B 0.000, C 0.000 }
gfCNCPoint5[7744] = {X 192.7625, Y 35.1971, Z -7.1667, A 0.000, B 0.000, C 0.000 }
gfCNCPoint5[7745] = {X 192.9743, Y 34.4796, Z -7.1667, A 0.000, B 0.000, C 0.000 }
gfCNCPoint5[7746] = {X 193.3110, Y 33.8117, Z -7.1667, A 0.000, B 0.000, C 0.000 }
gfCNCPoint5[7747] = {X 192.6982, Y 33.9570, Z -7.1667, A 0.000, B 0.000, C 0.000 }
gfCNCPoint5[7748] = {X 190.9622, Y 34.2317, Z -7.1667, A 0.000, B 0.000, C 0.000 }
gfCNCPoint5[7749] = {X 189.2131, Y 34.4056, Z -7.1667, A 0.000, B 0.000, C 0.000 }
gfCNCPoint5[7750] = {X 186.9480, Y 34.5447, Z -7.1667, A 0.000, B 0.000, C 0.000 }
gfCNCPoint5[7751] = {X 182.9921, Y 35.1369, Z -7.1667, A 0.000, B 0.000, C 0.000 }
gfCNCPoint5[7752] = {X 190.9418, Y 34.5686, Z -7.1667, A 0.000, B 0.000, C 0.000 }
gfCNCPoint5[7753] = {X 186.9431, Y 34.4648, Z -7.1667, A 0.000, B 0.000, C 0.000 }
gfCNCPoint5[7754] = {X 182.5719, Y 34.7332, Z -7.1667, A 0.000, B 0.000, C 0.000 }
gfCNCPoint5[7755] = {X 181.6836, Y 34.8406, Z -7.1667, A 0.000, B 0.000, C 0.000 }
gfCNCPoint5[7756] = {X 180.8142, Y 35.0516, Z -7.1667, A 0.000, B 0.000, C 0.000 }
gfCNCPoint5[7757] = {X 180.7587, Y 35.2519, Z -7.1667, A 0.000, B 0.000, C 0.000 }
gfCNCPoint5[7758] = {X 180.7458, Y 35.4593, Z -7.1667, A 0.000, B 0.000, C 0.000 }
gfCNCPoint5[7759] = {X 180.8554, Y 36.1029, Z -7.1667, A 0.000, B 0.000, C 0.000 }
gfCNCPoint5[7760] = {X 181.1604, Y 36.6802, Z -7.1667, A 0.000, B 0.000, C 0.000 }
gfCNCPoint5[7761] = {X 181.6303, Y 37.1334, Z -7.1667, A 0.000, B 0.000, C 0.000 }
gfCNCPoint5[7762] = {X 182.2892, Y 37.5103, Z -7.1667, A 0.000, B 0.000, C 0.000 }
gfCNCPoint5[7763] = {X 182.9939, Y 37.7922, Z -7.1667, A 0.000, B 0.000, C 0.000 }
gfCNCPoint5[7764] = {X 184.4482, Y 38.1170, Z -7.1667, A 0.000, B 0.000, C 0.000 }
gfCNCPoint5[7765] = {X 185.9336, Y 38.2363, Z -7.1667, A 0.000, B 0.000, C 0.000 }
gfCNCPoint5[7766] = {X 187.4212, Y 38.1479, Z -7.1667, A 0.000, B 0.000, C 0.000 }
gfCNCPoint5[7767] = {X 188.8820, Y 37.8534, Z -7.1667, A 0.000, B 0.000, C 0.000 }
gfCNCPoint5[7768] = {X 190.2876, Y 37.3587, Z -7.1667, A 0.000, B 0.000, C 0.000 }
gfCNCPoint5[7769] = {X 191.5591, Y 36.7323, Z -7.1667, A 0.000, B 0.000, C 0.000 }
gfCNCPoint5[7770] = {X 192.7622, Y 35.9832, Z -7.1667, A 0.000, B 0.000, C 0.000 }
gfCNCPoint5[7771] = {X 192.8357, Y 35.2395, Z -7.1667, A 0.000, B 0.000, C 0.000 }
gfCNCPoint5[7772] = {X 193.0436, Y 34.5218, Z -7.1667, A 0.000, B 0.000, C 0.000 }
gfCNCPoint5[7773] = {X 193.3790, Y 33.8540, Z -7.1667, A 0.000, B 0.000, C 0.000 }
gfCNCPoint5[7774] = {X 193.4221, Y 33.7861, Z -7.1667, A 0.000, B 0.000, C 0.000 }
gfCNCPoint5[7775] = {X 193.4667, Y 33.7192, Z -7.1667, A 0.000, B 0.000, C 0.000 }
gfCNCPoint5[7776] = {X 193.3658, Y 33.7165, Z -7.1667, A 0.000, B 0.000, C 0.000 }
gfCNCPoint5[7777] = {X 192.6816, Y 33.8787, Z -7.1667, A 0.000, B 0.000, C 0.000 }
gfCNCPoint5[7778] = {X 190.9512, Y 34.1525, Z -7.1667, A 0.000, B 0.000, C 0.000 }
gfCNCPoint5[7779] = {X 189.2078, Y 34.3258, Z -7.1667, A 0.000, B 0.000, C 0.000 }
gfCNCPoint5[7780] = {X 186.9431, Y 34.4648, Z -7.1667, A 0.000, B 0.000, C 0.000 }
gfCNCPoint5[7781] = {X 182.9872, Y 35.0570, Z -7.1667, A 0.000, B 0.000, C 0.000 }
gfCNCPoint5[7782] = {X 190.9369, Y 34.4887, Z -7.1667, A 0.000, B 0.000, C 0.000 }
gfCNCPoint5[7783] = {X 186.9382, Y 34.3850, Z -7.1667, A 0.000, B 0.000, C 0.000 }
gfCNCPoint5[7784] = {X 182.5670, Y 34.6534, Z -7.1667, A 0.000, B 0.000, C 0.000 }
gfCNCPoint5[7785] = {X 181.6508, Y 34.7652, Z -7.1667, A 0.000, B 0.000, C 0.000 }
gfCNCPoint5[7786] = {X 180.7547, Y 34.9863, Z -7.1667, A 0.000, B 0.000, C 0.000 }
gfCNCPoint5[7787] = {X 180.6833, Y 35.2188, Z -7.1667, A 0.000, B 0.000, C 0.000 }
gfCNCPoint5[7788] = {X 180.6658, Y 35.4613, Z -7.1667, A 0.000, B 0.000, C 0.000 }
gfCNCPoint5[7789] = {X 180.7800, Y 36.1297, Z -7.1667, A 0.000, B 0.000, C 0.000 }
gfCNCPoint5[7790] = {X 181.0970, Y 36.7290, Z -7.1667, A 0.000, B 0.000, C 0.000 }
gfCNCPoint5[7791] = {X 181.5852, Y 37.1995, Z -7.1667, A 0.000, B 0.000, C 0.000 }
gfCNCPoint5[7792] = {X 182.2544, Y 37.5823, Z -7.1667, A 0.000, B 0.000, C 0.000 }
gfCNCPoint5[7793] = {X 182.9702, Y 37.8686, Z -7.1667, A 0.000, B 0.000, C 0.000 }
gfCNCPoint5[7794] = {X 184.4356, Y 38.1960, Z -7.1667, A 0.000, B 0.000, C 0.000 }
gfCNCPoint5[7795] = {X 185.9323, Y 38.3163, Z -7.1667, A 0.000, B 0.000, C 0.000 }
gfCNCPoint5[7796] = {X 187.4311, Y 38.2273, Z -7.1667, A 0.000, B 0.000, C 0.000 }
gfCNCPoint5[7797] = {X 188.9031, Y 37.9306, Z -7.1667, A 0.000, B 0.000, C 0.000 }
gfCNCPoint5[7798] = {X 190.3194, Y 37.4321, Z -7.1667, A 0.000, B 0.000, C 0.000 }
gfCNCPoint5[7799] = {X 191.6162, Y 36.7921, Z -7.1667, A 0.000, B 0.000, C 0.000 }
gfCNCPoint5[7800] = {X 192.8422, Y 36.0250, Z -7.1667, A 0.000, B 0.000, C 0.000 }
gfCNCPoint5[7801] = {X 192.9290, Y 35.1818, Z -7.1667, A 0.000, B 0.000, C 0.000 }
gfCNCPoint5[7802] = {X 193.1917, Y 34.3757, Z -7.1667, A 0.000, B 0.000, C 0.000 }
gfCNCPoint5[7803] = {X 193.6183, Y 33.6431, Z -7.1667, A 0.000, B 0.000, C 0.000 }
gfCNCPoint5[7804] = {X 193.3575, Y 33.6362, Z -7.1667, A 0.000, B 0.000, C 0.000 }
gfCNCPoint5[7805] = {X 192.6650, Y 33.8004, Z -7.1667, A 0.000, B 0.000, C 0.000 }
gfCNCPoint5[7806] = {X 190.9402, Y 34.0732, Z -7.1667, A 0.000, B 0.000, C 0.000 }
gfCNCPoint5[7807] = {X 189.2026, Y 34.2460, Z -7.1667, A 0.000, B 0.000, C 0.000 }
gfCNCPoint5[7808] = {X 186.9382, Y 34.3850, Z -7.1667, A 0.000, B 0.000, C 0.000 }
gfCNCPoint5[7809] = {X 182.9823, Y 34.9772, Z -7.1667, A 0.000, B 0.000, C 0.000 }
gfCNCPoint5[7810] = {X 182.9823, Y 34.9772, Z -4.1667, A 0.000, B 0.000, C 0.000 }
gfCNCPoint5[7811] = {X 182.9823, Y 34.9772, Z 11.0000, A 0.000, B 0.000, C 0.000 }
gfCNCPoint5[7812] = {X 188.4995, Y 19.4688, Z 11.0000, A 0.000, B 0.000, C 0.000 }
gfCNCPoint5[7813] = {X 188.4995, Y 19.4688, Z -3.3333, A 0.000, B 0.000, C 0.000 }
gfCNCPoint5[7814] = {X 188.3884, Y 19.4295, Z -3.3649, A 0.000, B 0.000, C 0.000 }
gfCNCPoint5[7815] = {X 187.7714, Y 19.3609, Z -3.5313, A 0.000, B 0.000, C 0.000 }
gfCNCPoint5[7816] = {X 186.9109, Y 19.2609, Z -3.7634, A 0.000, B 0.000, C 0.000 }
gfCNCPoint5[7817] = {X 184.5930, Y 19.3684, Z -4.3851, A 0.000, B 0.000, C 0.000 }
gfCNCPoint5[7818] = {X 183.7426, Y 19.5482, Z -4.6180, A 0.000, B 0.000, C 0.000 }
gfCNCPoint5[7819] = {X 183.0434, Y 19.6907, Z -4.8092, A 0.000, B 0.000, C 0.000 }
gfCNCPoint5[7820] = {X 182.0226, Y 20.0622, Z -5.1003, A 0.000, B 0.000, C 0.000 }
gfCNCPoint5[7821] = {X 181.3954, Y 20.4024, Z -5.2915, A 0.000, B 0.000, C 0.000 }
gfCNCPoint5[7822] = {X 181.3393, Y 20.9140, Z -5.4294, A 0.000, B 0.000, C 0.000 }
gfCNCPoint5[7823] = {X 180.8654, Y 22.1252, Z -5.7779, A 0.000, B 0.000, C 0.000 }
gfCNCPoint5[7824] = {X 180.5594, Y 22.5391, Z -5.9158, A 0.000, B 0.000, C 0.000 }
gfCNCPoint5[7825] = {X 182.2921, Y 22.3331, Z -6.3834, A 0.000, B 0.000, C 0.000 }
gfCNCPoint5[7826] = {X 182.5945, Y 22.3086, Z -6.4646, A 0.000, B 0.000, C 0.000 }
gfCNCPoint5[7827] = {X 184.3413, Y 22.2325, Z -6.9331, A 0.000, B 0.000, C 0.000 }
gfCNCPoint5[7828] = {X 184.7768, Y 22.2173, Z -7.0499, A 0.000, B 0.000, C 0.000 }
gfCNCPoint5[7829] = {X 185.2122, Y 22.1989, Z -7.1667, A 0.000, B 0.000, C 0.000 }
gfCNCPoint5[7830] = {X 187.5423, Y 22.0765, Z -7.1667, A 0.000, B 0.000, C 0.000 }
gfCNCPoint5[7831] = {X 189.8694, Y 21.9068, Z -7.1667, A 0.000, B 0.000, C 0.000 }
gfCNCPoint5[7832] = {X 190.4708, Y 21.8301, Z -7.1667, A 0.000, B 0.000, C 0.000 }
gfCNCPoint5[7833] = {X 191.0578, Y 21.6789, Z -7.1667, A 0.000, B 0.000, C 0.000 }
gfCNCPoint5[7834] = {X 191.0675, Y 21.1637, Z -7.1667, A 0.000, B 0.000, C 0.000 }
gfCNCPoint5[7835] = {X 190.8719, Y 20.6870, Z -7.1667, A 0.000, B 0.000, C 0.000 }
gfCNCPoint5[7836] = {X 190.5032, Y 20.3270, Z -7.1667, A 0.000, B 0.000, C 0.000 }
gfCNCPoint5[7837] = {X 189.6457, Y 19.8663, Z -7.1667, A 0.000, B 0.000, C 0.000 }
gfCNCPoint5[7838] = {X 188.7279, Y 19.5418, Z -7.1667, A 0.000, B 0.000, C 0.000 }
gfCNCPoint5[7839] = {X 187.7714, Y 19.3609, Z -7.1667, A 0.000, B 0.000, C 0.000 }
gfCNCPoint5[7840] = {X 186.4243, Y 19.2778, Z -7.1667, A 0.000, B 0.000, C 0.000 }
gfCNCPoint5[7841] = {X 185.0761, Y 19.3405, Z -7.1667, A 0.000, B 0.000, C 0.000 }
gfCNCPoint5[7842] = {X 183.7426, Y 19.5482, Z -7.1667, A 0.000, B 0.000, C 0.000 }
gfCNCPoint5[7843] = {X 182.5373, Y 19.8883, Z -7.1667, A 0.000, B 0.000, C 0.000 }
gfCNCPoint5[7844] = {X 181.3954, Y 20.4024, Z -7.1667, A 0.000, B 0.000, C 0.000 }
gfCNCPoint5[7845] = {X 181.2441, Y 21.1602, Z -7.1667, A 0.000, B 0.000, C 0.000 }
gfCNCPoint5[7846] = {X 180.9625, Y 21.8798, Z -7.1667, A 0.000, B 0.000, C 0.000 }
gfCNCPoint5[7847] = {X 180.5594, Y 22.5391, Z -7.1667, A 0.000, B 0.000, C 0.000 }
gfCNCPoint5[7848] = {X 182.4475, Y 22.3504, Z -7.1667, A 0.000, B 0.000, C 0.000 }
gfCNCPoint5[7849] = {X 184.3413, Y 22.2325, Z -7.1667, A 0.000, B 0.000, C 0.000 }
gfCNCPoint5[7850] = {X 184.7768, Y 22.2165, Z -7.1667, A 0.000, B 0.000, C 0.000 }
gfCNCPoint5[7851] = {X 185.2122, Y 22.1989, Z -7.1667, A 0.000, B 0.000, C 0.000 }
gfCNCPoint5[7852] = {X 181.2196, Y 22.0991, Z -7.1667, A 0.000, B 0.000, C 0.000 }
gfCNCPoint5[7853] = {X 185.2156, Y 22.2788, Z -7.1667, A 0.000, B 0.000, C 0.000 }
gfCNCPoint5[7854] = {X 187.5450, Y 22.1565, Z -7.1667, A 0.000, B 0.000, C 0.000 }
gfCNCPoint5[7855] = {X 189.8716, Y 21.9868, Z -7.1667, A 0.000, B 0.000, C 0.000 }
gfCNCPoint5[7856] = {X 190.5063, Y 21.9047, Z -7.1667, A 0.000, B 0.000, C 0.000 }
gfCNCPoint5[7857] = {X 191.1250, Y 21.7410, Z -7.1667, A 0.000, B 0.000, C 0.000 }
gfCNCPoint5[7858] = {X 191.1514, Y 21.1790, Z -7.1667, A 0.000, B 0.000, C 0.000 }
gfCNCPoint5[7859] = {X 190.9467, Y 20.6549, Z -7.1667, A 0.000, B 0.000, C 0.000 }
gfCNCPoint5[7860] = {X 190.5464, Y 20.2596, Z -7.1667, A 0.000, B 0.000, C 0.000 }
gfCNCPoint5[7861] = {X 189.6787, Y 19.7934, Z -7.1667, A 0.000, B 0.000, C 0.000 }
gfCNCPoint5[7862] = {X 188.7501, Y 19.4649, Z -7.1667, A 0.000, B 0.000, C 0.000 }
gfCNCPoint5[7863] = {X 187.7823, Y 19.2816, Z -7.1667, A 0.000, B 0.000, C 0.000 }
gfCNCPoint5[7864] = {X 186.4270, Y 19.1978, Z -7.1667, A 0.000, B 0.000, C 0.000 }
gfCNCPoint5[7865] = {X 185.0706, Y 19.2606, Z -7.1667, A 0.000, B 0.000, C 0.000 }
gfCNCPoint5[7866] = {X 183.7289, Y 19.4693, Z -7.1667, A 0.000, B 0.000, C 0.000 }
gfCNCPoint5[7867] = {X 182.4919, Y 19.8197, Z -7.1667, A 0.000, B 0.000, C 0.000 }
gfCNCPoint5[7868] = {X 181.3215, Y 20.3516, Z -7.1667, A 0.000, B 0.000, C 0.000 }
gfCNCPoint5[7869] = {X 181.1583, Y 21.1711, Z -7.1667, A 0.000, B 0.000, C 0.000 }
gfCNCPoint5[7870] = {X 180.8403, Y 21.9439, Z -7.1667, A 0.000, B 0.000, C 0.000 }
gfCNCPoint5[7871] = {X 180.3795, Y 22.6409, Z -7.1667, A 0.000, B 0.000, C 0.000 }
gfCNCPoint5[7872] = {X 182.3578, Y 22.4378, Z -7.1667, A 0.000, B 0.000, C 0.000 }
gfCNCPoint5[7873] = {X 184.3427, Y 22.3125, Z -7.1667, A 0.000, B 0.000, C 0.000 }
gfCNCPoint5[7874] = {X 184.7791, Y 22.2965, Z -7.1667, A 0.000, B 0.000, C 0.000 }
gfCNCPoint5[7875] = {X 185.2156, Y 22.2788, Z -7.1667, A 0.000, B 0.000, C 0.000 }
gfCNCPoint5[7876] = {X 189.1820, Y 21.7619, Z -7.1667, A 0.000, B 0.000, C 0.000 }
gfCNCPoint5[7877] = {X 181.2230, Y 22.1791, Z -7.1667, A 0.000, B 0.000, C 0.000 }
gfCNCPoint5[7878] = {X 185.2189, Y 22.3588, Z -7.1667, A 0.000, B 0.000, C 0.000 }
gfCNCPoint5[7879] = {X 187.5497, Y 22.2363, Z -7.1667, A 0.000, B 0.000, C 0.000 }
gfCNCPoint5[7880] = {X 189.8774, Y 22.0666, Z -7.1667, A 0.000, B 0.000, C 0.000 }
gfCNCPoint5[7881] = {X 190.5429, Y 21.9790, Z -7.1667, A 0.000, B 0.000, C 0.000 }
gfCNCPoint5[7882] = {X 191.1907, Y 21.8031, Z -7.1667, A 0.000, B 0.000, C 0.000 }
gfCNCPoint5[7883] = {X 191.2484, Y 21.3476, Z -7.1667, A 0.000, B 0.000, C 0.000 }
gfCNCPoint5[7884] = {X 191.1589, Y 20.8974, Z -7.1667, A 0.000, B 0.000, C 0.000 }
gfCNCPoint5[7885] = {X 190.9315, Y 20.4985, Z -7.1667, A 0.000, B 0.000, C 0.000 }
gfCNCPoint5[7886] = {X 190.5895, Y 20.1922, Z -7.1667, A 0.000, B 0.000, C 0.000 }
gfCNCPoint5[7887] = {X 189.7110, Y 19.7203, Z -7.1667, A 0.000, B 0.000, C 0.000 }
gfCNCPoint5[7888] = {X 188.7709, Y 19.3876, Z -7.1667, A 0.000, B 0.000, C 0.000 }
gfCNCPoint5[7889] = {X 187.7911, Y 19.2021, Z -7.1667, A 0.000, B 0.000, C 0.000 }
gfCNCPoint5[7890] = {X 186.4273, Y 19.1178, Z -7.1667, A 0.000, B 0.000, C 0.000 }
gfCNCPoint5[7891] = {X 185.0625, Y 19.1810, Z -7.1667, A 0.000, B 0.000, C 0.000 }
gfCNCPoint5[7892] = {X 183.7123, Y 19.3911, Z -7.1667, A 0.000, B 0.000, C 0.000 }
gfCNCPoint5[7893] = {X 182.4465, Y 19.7512, Z -7.1667, A 0.000, B 0.000, C 0.000 }
gfCNCPoint5[7894] = {X 181.2501, Y 20.2996, Z -7.1667, A 0.000, B 0.000, C 0.000 }
gfCNCPoint5[7895] = {X 181.2397, Y 20.3532, Z -7.1667, A 0.000, B 0.000, C 0.000 }
gfCNCPoint5[7896] = {X 181.0587, Y 21.2188, Z -7.1667, A 0.000, B 0.000, C 0.000 }
gfCNCPoint5[7897] = {X 180.7021, Y 22.0281, Z -7.1667, A 0.000, B 0.000, C 0.000 }
gfCNCPoint5[7898] = {X 180.1854, Y 22.7457, Z -7.1667, A 0.000, B 0.000, C 0.000 }
gfCNCPoint5[7899] = {X 182.2620, Y 22.5261, Z -7.1667, A 0.000, B 0.000, C 0.000 }
gfCNCPoint5[7900] = {X 184.3458, Y 22.3924, Z -7.1667, A 0.000, B 0.000, C 0.000 }
gfCNCPoint5[7901] = {X 184.7824, Y 22.3764, Z -7.1667, A 0.000, B 0.000, C 0.000 }
gfCNCPoint5[7902] = {X 185.2189, Y 22.3588, Z -7.1667, A 0.000, B 0.000, C 0.000 }
gfCNCPoint5[7903] = {X 189.1854, Y 21.8419, Z -7.1667, A 0.000, B 0.000, C 0.000 }
gfCNCPoint5[7904] = {X 181.2264, Y 22.2590, Z -7.1667, A 0.000, B 0.000, C 0.000 }
gfCNCPoint5[7905] = {X 185.2223, Y 22.4387, Z -7.1667, A 0.000, B 0.000, C 0.000 }
gfCNCPoint5[7906] = {X 187.5543, Y 22.3162, Z -7.1667, A 0.000, B 0.000, C 0.000 }
gfCNCPoint5[7907] = {X 189.8833, Y 22.1464, Z -7.1667, A 0.000, B 0.000, C 0.000 }
gfCNCPoint5[7908] = {X 190.5790, Y 22.0533, Z -7.1667, A 0.000, B 0.000, C 0.000 }
gfCNCPoint5[7909] = {X 191.2552, Y 21.8653, Z -7.1667, A 0.000, B 0.000, C 0.000 }
gfCNCPoint5[7910] = {X 191.3291, Y 21.3759, Z -7.1667, A 0.000, B 0.000, C 0.000 }
gfCNCPoint5[7911] = {X 191.2409, Y 20.8888, Z -7.1667, A 0.000, B 0.000, C 0.000 }
gfCNCPoint5[7912] = {X 191.0002, Y 20.4564, Z -7.1667, A 0.000, B 0.000, C 0.000 }
gfCNCPoint5[7913] = {X 190.6326, Y 20.1248, Z -7.1667, A 0.000, B 0.000, C 0.000 }
gfCNCPoint5[7914] = {X 189.7434, Y 19.6471, Z -7.1667, A 0.000, B 0.000, C 0.000 }
gfCNCPoint5[7915] = {X 188.7918, Y 19.3104, Z -7.1667, A 0.000, B 0.000, C 0.000 }
gfCNCPoint5[7916] = {X 187.7999, Y 19.1226, Z -7.1667, A 0.000, B 0.000, C 0.000 }
gfCNCPoint5[7917] = {X 186.4277, Y 19.0378, Z -7.1667, A 0.000, B 0.000, C 0.000 }
gfCNCPoint5[7918] = {X 185.0543, Y 19.1015, Z -7.1667, A 0.000, B 0.000, C 0.000 }
gfCNCPoint5[7919] = {X 183.6958, Y 19.3128, Z -7.1667, A 0.000, B 0.000, C 0.000 }
gfCNCPoint5[7920] = {X 182.4010, Y 19.6827, Z -7.1667, A 0.000, B 0.000, C 0.000 }
gfCNCPoint5[7921] = {X 181.1787, Y 20.2478, Z -7.1667, A 0.000, B 0.000, C 0.000 }
gfCNCPoint5[7922] = {X 181.1605, Y 20.3415, Z -7.1667, A 0.000, B 0.000, C 0.000 }
gfCNCPoint5[7923] = {X 180.9651, Y 21.2476, Z -7.1667, A 0.000, B 0.000, C 0.000 }
gfCNCPoint5[7924] = {X 180.5739, Y 22.0879, Z -7.1667, A 0.000, B 0.000, C 0.000 }
gfCNCPoint5[7925] = {X 180.0064, Y 22.8207, Z -7.1667, A 0.000, B 0.000, C 0.000 }
gfCNCPoint5[7926] = {X 180.1924, Y 22.8260, Z -7.1667, A 0.000, B 0.000, C 0.000 }
gfCNCPoint5[7927] = {X 182.2670, Y 22.6062, Z -7.1667, A 0.000, B 0.000, C 0.000 }
gfCNCPoint5[7928] = {X 184.3489, Y 22.4724, Z -7.1667, A 0.000, B 0.000, C 0.000 }
gfCNCPoint5[7929] = {X 184.7857, Y 22.4564, Z -7.1667, A 0.000, B 0.000, C 0.000 }
gfCNCPoint5[7930] = {X 185.2223, Y 22.4387, Z -7.1667, A 0.000, B 0.000, C 0.000 }
gfCNCPoint5[7931] = {X 189.1888, Y 21.9218, Z -7.1667, A 0.000, B 0.000, C 0.000 }
gfCNCPoint5[7932] = {X 181.2298, Y 22.3389, Z -7.1667, A 0.000, B 0.000, C 0.000 }
gfCNCPoint5[7933] = {X 185.2257, Y 22.5186, Z -7.1667, A 0.000, B 0.000, C 0.000 }
gfCNCPoint5[7934] = {X 187.5589, Y 22.3961, Z -7.1667, A 0.000, B 0.000, C 0.000 }
gfCNCPoint5[7935] = {X 189.8892, Y 22.2262, Z -7.1667, A 0.000, B 0.000, C 0.000 }
gfCNCPoint5[7936] = {X 190.6145, Y 22.1277, Z -7.1667, A 0.000, B 0.000, C 0.000 }
gfCNCPoint5[7937] = {X 191.3186, Y 21.9276, Z -7.1667, A 0.000, B 0.000, C 0.000 }
gfCNCPoint5[7938] = {X 191.4092, Y 21.4045, Z -7.1667, A 0.000, B 0.000, C 0.000 }
gfCNCPoint5[7939] = {X 191.3228, Y 20.8806, Z -7.1667, A 0.000, B 0.000, C 0.000 }
gfCNCPoint5[7940] = {X 191.0689, Y 20.4143, Z -7.1667, A 0.000, B 0.000, C 0.000 }
gfCNCPoint5[7941] = {X 190.6758, Y 20.0575, Z -7.1667, A 0.000, B 0.000, C 0.000 }
gfCNCPoint5[7942] = {X 189.7758, Y 19.5739, Z -7.1667, A 0.000, B 0.000, C 0.000 }
gfCNCPoint5[7943] = {X 188.8126, Y 19.2332, Z -7.1667, A 0.000, B 0.000, C 0.000 }
gfCNCPoint5[7944] = {X 187.8088, Y 19.0431, Z -7.1667, A 0.000, B 0.000, C 0.000 }
gfCNCPoint5[7945] = {X 186.4280, Y 18.9578, Z -7.1667, A 0.000, B 0.000, C 0.000 }
gfCNCPoint5[7946] = {X 185.0462, Y 19.0219, Z -7.1667, A 0.000, B 0.000, C 0.000 }
gfCNCPoint5[7947] = {X 183.6792, Y 19.2345, Z -7.1667, A 0.000, B 0.000, C 0.000 }
gfCNCPoint5[7948] = {X 182.3554, Y 19.6143, Z -7.1667, A 0.000, B 0.000, C 0.000 }
gfCNCPoint5[7949] = {X 181.1072, Y 20.1963, Z -7.1667, A 0.000, B 0.000, C 0.000 }
gfCNCPoint5[7950] = {X 181.0812, Y 20.3299, Z -7.1667, A 0.000, B 0.000, C 0.000 }
gfCNCPoint5[7951] = {X 180.8699, Y 21.2784, Z -7.1667, A 0.000, B 0.000, C 0.000 }
gfCNCPoint5[7952] = {X 180.4402, Y 22.1500, Z -7.1667, A 0.000, B 0.000, C 0.000 }
gfCNCPoint5[7953] = {X 179.8166, Y 22.8953, Z -7.1667, A 0.000, B 0.000, C 0.000 }
gfCNCPoint5[7954] = {X 180.1963, Y 22.9061, Z -7.1667, A 0.000, B 0.000, C 0.000 }
gfCNCPoint5[7955] = {X 182.2705, Y 22.6862, Z -7.1667, A 0.000, B 0.000, C 0.000 }
gfCNCPoint5[7956] = {X 184.3520, Y 22.5523, Z -7.1667, A 0.000, B 0.000, C 0.000 }
gfCNCPoint5[7957] = {X 184.7889, Y 22.5363, Z -7.1667, A 0.000, B 0.000, C 0.000 }
gfCNCPoint5[7958] = {X 185.2257, Y 22.5186, Z -7.1667, A 0.000, B 0.000, C 0.000 }
gfCNCPoint5[7959] = {X 189.1922, Y 22.0017, Z -7.1667, A 0.000, B 0.000, C 0.000 }
gfCNCPoint5[7960] = {X 185.1541, Y 22.6017, Z -7.1667, A 0.000, B 0.000, C 0.000 }
gfCNCPoint5[7961] = {X 185.2291, Y 22.5986, Z -7.1667, A 0.000, B 0.000, C 0.000 }
gfCNCPoint5[7962] = {X 187.5636, Y 22.4759, Z -7.1667, A 0.000, B 0.000, C 0.000 }
gfCNCPoint5[7963] = {X 189.8950, Y 22.3060, Z -7.1667, A 0.000, B 0.000, C 0.000 }
gfCNCPoint5[7964] = {X 190.6495, Y 22.2021, Z -7.1667, A 0.000, B 0.000, C 0.000 }
gfCNCPoint5[7965] = {X 191.3809, Y 21.9899, Z -7.1667, A 0.000, B 0.000, C 0.000 }
gfCNCPoint5[7966] = {X 191.4889, Y 21.4333, Z -7.1667, A 0.000, B 0.000, C 0.000 }
gfCNCPoint5[7967] = {X 191.4046, Y 20.8726, Z -7.1667, A 0.000, B 0.000, C 0.000 }
gfCNCPoint5[7968] = {X 191.1377, Y 20.3724, Z -7.1667, A 0.000, B 0.000, C 0.000 }
gfCNCPoint5[7969] = {X 190.7189, Y 19.9901, Z -7.1667, A 0.000, B 0.000, C 0.000 }
gfCNCPoint5[7970] = {X 189.8081, Y 19.5008, Z -7.1667, A 0.000, B 0.000, C 0.000 }
gfCNCPoint5[7971] = {X 188.8334, Y 19.1559, Z -7.1667, A 0.000, B 0.000, C 0.000 }
gfCNCPoint5[7972] = {X 187.8176, Y 18.9636, Z -7.1667, A 0.000, B 0.000, C 0.000 }
gfCNCPoint5[7973] = {X 186.4284, Y 18.8778, Z -7.1667, A 0.000, B 0.000, C 0.000 }
gfCNCPoint5[7974] = {X 185.0380, Y 18.9423, Z -7.1667, A 0.000, B 0.000, C 0.000 }
gfCNCPoint5[7975] = {X 183.6627, Y 19.1563, Z -7.1667, A 0.000, B 0.000, C 0.000 }
gfCNCPoint5[7976] = {X 182.3098, Y 19.5460, Z -7.1667, A 0.000, B 0.000, C 0.000 }
gfCNCPoint5[7977] = {X 181.0357, Y 20.1449, Z -7.1667, A 0.000, B 0.000, C 0.000 }
gfCNCPoint5[7978] = {X 181.0020, Y 20.3183, Z -7.1667, A 0.000, B 0.000, C 0.000 }
gfCNCPoint5[7979] = {X 180.8538, Y 21.0695, Z -7.1667, A 0.000, B 0.000, C 0.000 }
gfCNCPoint5[7980] = {X 180.5651, Y 21.7787, Z -7.1667, A 0.000, B 0.000, C 0.000 }
gfCNCPoint5[7981] = {X 180.1466, Y 22.4199, Z -7.1667, A 0.000, B 0.000, C 0.000 }
gfCNCPoint5[7982] = {X 179.6136, Y 22.9696, Z -7.1667, A 0.000, B 0.000, C 0.000 }
gfCNCPoint5[7983] = {X 180.2003, Y 22.9863, Z -7.1667, A 0.000, B 0.000, C 0.000 }
gfCNCPoint5[7984] = {X 182.2741, Y 22.7662, Z -7.1667, A 0.000, B 0.000, C 0.000 }
gfCNCPoint5[7985] = {X 184.3552, Y 22.6322, Z -7.1667, A 0.000, B 0.000, C 0.000 }
gfCNCPoint5[7986] = {X 184.7922, Y 22.6162, Z -7.1667, A 0.000, B 0.000, C 0.000 }
gfCNCPoint5[7987] = {X 185.2291, Y 22.5986, Z -7.1667, A 0.000, B 0.000, C 0.000 }
gfCNCPoint5[7988] = {X 185.1445, Y 20.6003, Z -7.1667, A 0.000, B 0.000, C 0.000 }
gfCNCPoint5[7989] = {X 185.1445, Y 20.6003, Z -4.1667, A 0.000, B 0.000, C 0.000 }
gfCNCPoint5[7990] = {X 185.1445, Y 20.6003, Z 11.0000, A 0.000, B 0.000, C 0.000 }
gfCNCPoint5[7991] = {X 256.2473, Y 19.7825, Z 11.0000, A 0.000, B 0.000, C 0.000 }
gfCNCPoint5[7992] = {X 256.2473, Y 19.7825, Z -3.3333, A 0.000, B 0.000, C 0.000 }
gfCNCPoint5[7993] = {X 251.5292, Y 19.7821, Z -4.5975, A 0.000, B 0.000, C 0.000 }
gfCNCPoint5[7994] = {X 250.8344, Y 19.7929, Z -4.7837, A 0.000, B 0.000, C 0.000 }
gfCNCPoint5[7995] = {X 250.1815, Y 19.7942, Z -4.9587, A 0.000, B 0.000, C 0.000 }
gfCNCPoint5[7996] = {X 249.4949, Y 19.8927, Z -5.1445, A 0.000, B 0.000, C 0.000 }
gfCNCPoint5[7997] = {X 248.8454, Y 20.0810, Z -5.3257, A 0.000, B 0.000, C 0.000 }
gfCNCPoint5[7998] = {X 248.7087, Y 20.1123, Z -5.3633, A 0.000, B 0.000, C 0.000 }
gfCNCPoint5[7999] = {X 248.6551, Y 20.1625, Z -5.3830, A 0.000, B 0.000, C 0.000 }
gfCNCPoint5[8000] = {X 248.6152, Y 20.2970, Z -5.4206, A 0.000, B 0.000, C 0.000 }
gfCNCPoint5[8001] = {X 248.4762, Y 20.7653, Z -5.5515, A 0.000, B 0.000, C 0.000 }
gfCNCPoint5[8002] = {X 248.4460, Y 21.8665, Z -5.8467, A 0.000, B 0.000, C 0.000 }
gfCNCPoint5[8003] = {X 248.5591, Y 22.3418, Z -5.9775, A 0.000, B 0.000, C 0.000 }
gfCNCPoint5[8004] = {X 248.8765, Y 22.4371, Z -6.0663, A 0.000, B 0.000, C 0.000 }
gfCNCPoint5[8005] = {X 249.2069, Y 22.4640, Z -6.1551, A 0.000, B 0.000, C 0.000 }
gfCNCPoint5[8006] = {X 250.4436, Y 22.5649, Z -6.4876, A 0.000, B 0.000, C 0.000 }
gfCNCPoint5[8007] = {X 251.6873, Y 22.5560, Z -6.8209, A 0.000, B 0.000, C 0.000 }
gfCNCPoint5[8008] = {X 252.9778, Y 22.5560, Z -7.1667, A 0.000, B 0.000, C 0.000 }
gfCNCPoint5[8009] = {X 257.4115, Y 22.5560, Z -7.1667, A 0.000, B 0.000, C 0.000 }
gfCNCPoint5[8010] = {X 257.4115, Y 19.7825, Z -7.1667, A 0.000, B 0.000, C 0.000 }
gfCNCPoint5[8011] = {X 251.5292, Y 19.7821, Z -7.1667, A 0.000, B 0.000, C 0.000 }
gfCNCPoint5[8012] = {X 250.8344, Y 19.7929, Z -7.1667, A 0.000, B 0.000, C 0.000 }
gfCNCPoint5[8013] = {X 249.8297, Y 19.8661, Z -7.1667, A 0.000, B 0.000, C 0.000 }
gfCNCPoint5[8014] = {X 248.8454, Y 20.0810, Z -7.1667, A 0.000, B 0.000, C 0.000 }
gfCNCPoint5[8015] = {X 248.7011, Y 20.1578, Z -7.1667, A 0.000, B 0.000, C 0.000 }
gfCNCPoint5[8016] = {X 248.6152, Y 20.2970, Z -7.1667, A 0.000, B 0.000, C 0.000 }
gfCNCPoint5[8017] = {X 248.4774, Y 20.9718, Z -7.1667, A 0.000, B 0.000, C 0.000 }
gfCNCPoint5[8018] = {X 248.4585, Y 21.6604, Z -7.1667, A 0.000, B 0.000, C 0.000 }
gfCNCPoint5[8019] = {X 248.5591, Y 22.3418, Z -7.1667, A 0.000, B 0.000, C 0.000 }
gfCNCPoint5[8020] = {X 248.8798, Y 22.4199, Z -7.1667, A 0.000, B 0.000, C 0.000 }
gfCNCPoint5[8021] = {X 249.2069, Y 22.4640, Z -7.1667, A 0.000, B 0.000, C 0.000 }
gfCNCPoint5[8022] = {X 250.4461, Y 22.5375, Z -7.1667, A 0.000, B 0.000, C 0.000 }
gfCNCPoint5[8023] = {X 251.6873, Y 22.5560, Z -7.1667, A 0.000, B 0.000, C 0.000 }
gfCNCPoint5[8024] = {X 252.9778, Y 22.5560, Z -7.1667, A 0.000, B 0.000, C 0.000 }
gfCNCPoint5[8025] = {X 248.9930, Y 22.2874, Z -7.1667, A 0.000, B 0.000, C 0.000 }
gfCNCPoint5[8026] = {X 252.9778, Y 22.6360, Z -7.1667, A 0.000, B 0.000, C 0.000 }
gfCNCPoint5[8027] = {X 257.4915, Y 22.6360, Z -7.1667, A 0.000, B 0.000, C 0.000 }
gfCNCPoint5[8028] = {X 257.4915, Y 19.7026, Z -7.1667, A 0.000, B 0.000, C 0.000 }
gfCNCPoint5[8029] = {X 251.5286, Y 19.7021, Z -7.1667, A 0.000, B 0.000, C 0.000 }
gfCNCPoint5[8030] = {X 250.8364, Y 19.7129, Z -7.1667, A 0.000, B 0.000, C 0.000 }
gfCNCPoint5[8031] = {X 249.8259, Y 19.7862, Z -7.1667, A 0.000, B 0.000, C 0.000 }
gfCNCPoint5[8032] = {X 248.8357, Y 20.0012, Z -7.1667, A 0.000, B 0.000, C 0.000 }
gfCNCPoint5[8033] = {X 248.6494, Y 20.0966, Z -7.1667, A 0.000, B 0.000, C 0.000 }
gfCNCPoint5[8034] = {X 248.5385, Y 20.2742, Z -7.1667, A 0.000, B 0.000, C 0.000 }
gfCNCPoint5[8035] = {X 248.3962, Y 20.9779, Z -7.1667, A 0.000, B 0.000, C 0.000 }
gfCNCPoint5[8036] = {X 248.3806, Y 21.6957, Z -7.1667, A 0.000, B 0.000, C 0.000 }
gfCNCPoint5[8037] = {X 248.4922, Y 22.4048, Z -7.1667, A 0.000, B 0.000, C 0.000 }
gfCNCPoint5[8038] = {X 248.8424, Y 22.4942, Z -7.1667, A 0.000, B 0.000, C 0.000 }
gfCNCPoint5[8039] = {X 249.2003, Y 22.5438, Z -7.1667, A 0.000, B 0.000, C 0.000 }
gfCNCPoint5[8040] = {X 250.4422, Y 22.6174, Z -7.1667, A 0.000, B 0.000, C 0.000 }
gfCNCPoint5[8041] = {X 251.6862, Y 22.6360, Z -7.1667, A 0.000, B 0.000, C 0.000 }
gfCNCPoint5[8042] = {X 252.9778, Y 22.6360, Z -7.1667, A 0.000, B 0.000, C 0.000 }
gfCNCPoint5[8043] = {X 256.9625, Y 22.2874, Z -7.1667, A 0.000, B 0.000, C 0.000 }
gfCNCPoint5[8044] = {X 248.9930, Y 22.3674, Z -7.1667, A 0.000, B 0.000, C 0.000 }
gfCNCPoint5[8045] = {X 252.9778, Y 22.7160, Z -7.1667, A 0.000, B 0.000, C 0.000 }
gfCNCPoint5[8046] = {X 257.5715, Y 22.7160, Z -7.1667, A 0.000, B 0.000, C 0.000 }
gfCNCPoint5[8047] = {X 257.5715, Y 19.6226, Z -7.1667, A 0.000, B 0.000, C 0.000 }
gfCNCPoint5[8048] = {X 251.5280, Y 19.6221, Z -7.1667, A 0.000, B 0.000, C 0.000 }
gfCNCPoint5[8049] = {X 250.8357, Y 19.6329, Z -7.1667, A 0.000, B 0.000, C 0.000 }
gfCNCPoint5[8050] = {X 249.8156, Y 19.7068, Z -7.1667, A 0.000, B 0.000, C 0.000 }
gfCNCPoint5[8051] = {X 248.8161, Y 19.9236, Z -7.1667, A 0.000, B 0.000, C 0.000 }
gfCNCPoint5[8052] = {X 248.5940, Y 20.0389, Z -7.1667, A 0.000, B 0.000, C 0.000 }
gfCNCPoint5[8053] = {X 248.4618, Y 20.2515, Z -7.1667, A 0.000, B 0.000, C 0.000 }
gfCNCPoint5[8054] = {X 248.3151, Y 20.9838, Z -7.1667, A 0.000, B 0.000, C 0.000 }
gfCNCPoint5[8055] = {X 248.3029, Y 21.7306, Z -7.1667, A 0.000, B 0.000, C 0.000 }
gfCNCPoint5[8056] = {X 248.4256, Y 22.4674, Z -7.1667, A 0.000, B 0.000, C 0.000 }
gfCNCPoint5[8057] = {X 248.8051, Y 22.5683, Z -7.1667, A 0.000, B 0.000, C 0.000 }
gfCNCPoint5[8058] = {X 249.1938, Y 22.6235, Z -7.1667, A 0.000, B 0.000, C 0.000 }
gfCNCPoint5[8059] = {X 250.4391, Y 22.6974, Z -7.1667, A 0.000, B 0.000, C 0.000 }
gfCNCPoint5[8060] = {X 251.6865, Y 22.7160, Z -7.1667, A 0.000, B 0.000, C 0.000 }
gfCNCPoint5[8061] = {X 252.9778, Y 22.7160, Z -7.1667, A 0.000, B 0.000, C 0.000 }
gfCNCPoint5[8062] = {X 256.9625, Y 22.3674, Z -7.1667, A 0.000, B 0.000, C 0.000 }
gfCNCPoint5[8063] = {X 248.9930, Y 22.4474, Z -7.1667, A 0.000, B 0.000, C 0.000 }
gfCNCPoint5[8064] = {X 252.9778, Y 22.7960, Z -7.1667, A 0.000, B 0.000, C 0.000 }
gfCNCPoint5[8065] = {X 257.6515, Y 22.7960, Z -7.1667, A 0.000, B 0.000, C 0.000 }
gfCNCPoint5[8066] = {X 257.6515, Y 19.5426, Z -7.1667, A 0.000, B 0.000, C 0.000 }
gfCNCPoint5[8067] = {X 251.5274, Y 19.5421, Z -7.1667, A 0.000, B 0.000, C 0.000 }
gfCNCPoint5[8068] = {X 250.8350, Y 19.5529, Z -7.1667, A 0.000, B 0.000, C 0.000 }
gfCNCPoint5[8069] = {X 249.8053, Y 19.6275, Z -7.1667, A 0.000, B 0.000, C 0.000 }
gfCNCPoint5[8070] = {X 248.7963, Y 19.8460, Z -7.1667, A 0.000, B 0.000, C 0.000 }
gfCNCPoint5[8071] = {X 248.5385, Y 19.9813, Z -7.1667, A 0.000, B 0.000, C 0.000 }
gfCNCPoint5[8072] = {X 248.3851, Y 20.2287, Z -7.1667, A 0.000, B 0.000, C 0.000 }
gfCNCPoint5[8073] = {X 248.2340, Y 20.9896, Z -7.1667, A 0.000, B 0.000, C 0.000 }
gfCNCPoint5[8074] = {X 248.2253, Y 21.7653, Z -7.1667, A 0.000, B 0.000, C 0.000 }
gfCNCPoint5[8075] = {X 248.3594, Y 22.5294, Z -7.1667, A 0.000, B 0.000, C 0.000 }
gfCNCPoint5[8076] = {X 248.7679, Y 22.6424, Z -7.1667, A 0.000, B 0.000, C 0.000 }
gfCNCPoint5[8077] = {X 249.1873, Y 22.7032, Z -7.1667, A 0.000, B 0.000, C 0.000 }
gfCNCPoint5[8078] = {X 250.4360, Y 22.7773, Z -7.1667, A 0.000, B 0.000, C 0.000 }
gfCNCPoint5[8079] = {X 251.6868, Y 22.7960, Z -7.1667, A 0.000, B 0.000, C 0.000 }
gfCNCPoint5[8080] = {X 252.9778, Y 22.7960, Z -7.1667, A 0.000, B 0.000, C 0.000 }
gfCNCPoint5[8081] = {X 256.9625, Y 22.4474, Z -7.1667, A 0.000, B 0.000, C 0.000 }
gfCNCPoint5[8082] = {X 248.9930, Y 22.5274, Z -7.1667, A 0.000, B 0.000, C 0.000 }
gfCNCPoint5[8083] = {X 252.9778, Y 22.8760, Z -7.1667, A 0.000, B 0.000, C 0.000 }
gfCNCPoint5[8084] = {X 257.7315, Y 22.8760, Z -7.1667, A 0.000, B 0.000, C 0.000 }
gfCNCPoint5[8085] = {X 257.7315, Y 19.4626, Z -7.1667, A 0.000, B 0.000, C 0.000 }
gfCNCPoint5[8086] = {X 251.5267, Y 19.4621, Z -7.1667, A 0.000, B 0.000, C 0.000 }
gfCNCPoint5[8087] = {X 250.8343, Y 19.4729, Z -7.1667, A 0.000, B 0.000, C 0.000 }
gfCNCPoint5[8088] = {X 249.7949, Y 19.5482, Z -7.1667, A 0.000, B 0.000, C 0.000 }
gfCNCPoint5[8089] = {X 248.7763, Y 19.7685, Z -7.1667, A 0.000, B 0.000, C 0.000 }
gfCNCPoint5[8090] = {X 248.4830, Y 19.9237, Z -7.1667, A 0.000, B 0.000, C 0.000 }
gfCNCPoint5[8091] = {X 248.3084, Y 20.2059, Z -7.1667, A 0.000, B 0.000, C 0.000 }
gfCNCPoint5[8092] = {X 248.1537, Y 20.9889, Z -7.1667, A 0.000, B 0.000, C 0.000 }
gfCNCPoint5[8093] = {X 248.1469, Y 21.7870, Z -7.1667, A 0.000, B 0.000, C 0.000 }
gfCNCPoint5[8094] = {X 248.2883, Y 22.5725, Z -7.1667, A 0.000, B 0.000, C 0.000 }
gfCNCPoint5[8095] = {X 248.3069, Y 22.5959, Z -7.1667, A 0.000, B 0.000, C 0.000 }
gfCNCPoint5[8096] = {X 248.3333, Y 22.6051, Z -7.1667, A 0.000, B 0.000, C 0.000 }
gfCNCPoint5[8097] = {X 248.7515, Y 22.7206, Z -7.1667, A 0.000, B 0.000, C 0.000 }
gfCNCPoint5[8098] = {X 249.1808, Y 22.7830, Z -7.1667, A 0.000, B 0.000, C 0.000 }
gfCNCPoint5[8099] = {X 250.4329, Y 22.8572, Z -7.1667, A 0.000, B 0.000, C 0.000 }
gfCNCPoint5[8100] = {X 251.6870, Y 22.8760, Z -7.1667, A 0.000, B 0.000, C 0.000 }
gfCNCPoint5[8101] = {X 252.9778, Y 22.8760, Z -7.1667, A 0.000, B 0.000, C 0.000 }
gfCNCPoint5[8102] = {X 256.9625, Y 22.5274, Z -7.1667, A 0.000, B 0.000, C 0.000 }
gfCNCPoint5[8103] = {X 248.9930, Y 22.6074, Z -7.1667, A 0.000, B 0.000, C 0.000 }
gfCNCPoint5[8104] = {X 252.9778, Y 22.9560, Z -7.1667, A 0.000, B 0.000, C 0.000 }
gfCNCPoint5[8105] = {X 257.8115, Y 22.9560, Z -7.1667, A 0.000, B 0.000, C 0.000 }
gfCNCPoint5[8106] = {X 257.8115, Y 19.3826, Z -7.1667, A 0.000, B 0.000, C 0.000 }
gfCNCPoint5[8107] = {X 251.5261, Y 19.3821, Z -7.1667, A 0.000, B 0.000, C 0.000 }
gfCNCPoint5[8108] = {X 250.8336, Y 19.3929, Z -7.1667, A 0.000, B 0.000, C 0.000 }
gfCNCPoint5[8109] = {X 249.7844, Y 19.4689, Z -7.1667, A 0.000, B 0.000, C 0.000 }
gfCNCPoint5[8110] = {X 248.7562, Y 19.6911, Z -7.1667, A 0.000, B 0.000, C 0.000 }
gfCNCPoint5[8111] = {X 248.4274, Y 19.8661, Z -7.1667, A 0.000, B 0.000, C 0.000 }
gfCNCPoint5[8112] = {X 248.2317, Y 20.1832, Z -7.1667, A 0.000, B 0.000, C 0.000 }
gfCNCPoint5[8113] = {X 248.0735, Y 20.9862, Z -7.1667, A 0.000, B 0.000, C 0.000 }
gfCNCPoint5[8114] = {X 248.0681, Y 21.8046, Z -7.1667, A 0.000, B 0.000, C 0.000 }
gfCNCPoint5[8115] = {X 248.2156, Y 22.6097, Z -7.1667, A 0.000, B 0.000, C 0.000 }
gfCNCPoint5[8116] = {X 248.2586, Y 22.6635, Z -7.1667, A 0.000, B 0.000, C 0.000 }
gfCNCPoint5[8117] = {X 248.7098, Y 22.7936, Z -7.1667, A 0.000, B 0.000, C 0.000 }
gfCNCPoint5[8118] = {X 249.1743, Y 22.8627, Z -7.1667, A 0.000, B 0.000, C 0.000 }
gfCNCPoint5[8119] = {X 250.4298, Y 22.9372, Z -7.1667, A 0.000, B 0.000, C 0.000 }
gfCNCPoint5[8120] = {X 251.6873, Y 22.9560, Z -7.1667, A 0.000, B 0.000, C 0.000 }
gfCNCPoint5[8121] = {X 252.9778, Y 22.9560, Z -7.1667, A 0.000, B 0.000, C 0.000 }
gfCNCPoint5[8122] = {X 256.9625, Y 22.6074, Z -7.1667, A 0.000, B 0.000, C 0.000 }
gfCNCPoint5[8123] = {X 256.9625, Y 22.6074, Z -4.1667, A 0.000, B 0.000, C 0.000 }
gfCNCPoint5[8124] = {X 256.9625, Y 22.6074, Z 11.0000, A 0.000, B 0.000, C 0.000 }
gfCNCPoint5[8125] = {X 507.6812, Y 107.6951, Z 11.0000, A 0.000, B 0.000, C 0.000 }
gfCNCPoint5[8126] = {X 507.6812, Y 107.6951, Z -4.1667, A 0.000, B 0.000, C 0.000 }
gfCNCPoint5[8127] = {X 507.6812, Y 107.6951, Z -7.1667, A 0.000, B 0.000, C 0.000 }
gfCNCPoint5[8128] = {X 507.6812, Y 71.2951, Z -7.1667, A 0.000, B 0.000, C 0.000 }
gfCNCPoint5[8129] = {X 509.5505, Y 71.2951, Z -7.1667, A 0.000, B 0.000, C 0.000 }
gfCNCPoint5[8130] = {X 509.0280, Y 71.0692, Z -7.1667, A 0.000, B 0.000, C 0.000 }
gfCNCPoint5[8131] = {X 508.5105, Y 70.8320, Z -7.1667, A 0.000, B 0.000, C 0.000 }
gfCNCPoint5[8132] = {X 507.1672, Y 71.0985, Z -7.1667, A 0.000, B 0.000, C 0.000 }
gfCNCPoint5[8133] = {X 505.8120, Y 71.2951, Z -7.1667, A 0.000, B 0.000, C 0.000 }
gfCNCPoint5[8134] = {X 507.6812, Y 71.2951, Z -7.1667, A 0.000, B 0.000, C 0.000 }
gfCNCPoint5[8135] = {X 507.6812, Y 73.6951, Z -7.1667, A 0.000, B 0.000, C 0.000 }
gfCNCPoint5[8136] = {X 551.2537, Y 73.6951, Z -7.1667, A 0.000, B 0.000, C 0.000 }
gfCNCPoint5[8137] = {X 549.1244, Y 72.7708, Z -7.1667, A 0.000, B 0.000, C 0.000 }
gfCNCPoint5[8138] = {X 547.0707, Y 71.6888, Z -7.1667, A 0.000, B 0.000, C 0.000 }
gfCNCPoint5[8139] = {X 545.1043, Y 70.4552, Z -7.1667, A 0.000, B 0.000, C 0.000 }
gfCNCPoint5[8140] = {X 543.2365, Y 69.0769, Z -7.1667, A 0.000, B 0.000, C 0.000 }
gfCNCPoint5[8141] = {X 529.7627, Y 69.0772, Z -7.1667, A 0.000, B 0.000, C 0.000 }
gfCNCPoint5[8142] = {X 527.5498, Y 69.8803, Z -7.1667, A 0.000, B 0.000, C 0.000 }
gfCNCPoint5[8143] = {X 525.2695, Y 70.4649, Z -7.1667, A 0.000, B 0.000, C 0.000 }
gfCNCPoint5[8144] = {X 522.9432, Y 70.8256, Z -7.1667, A 0.000, B 0.000, C 0.000 }
gfCNCPoint5[8145] = {X 520.5929, Y 70.9589, Z -7.1667, A 0.000, B 0.000, C 0.000 }
gfCNCPoint5[8146] = {X 519.7998, Y 70.9591, Z -7.1667, A 0.000, B 0.000, C 0.000 }
gfCNCPoint5[8147] = {X 517.4111, Y 70.8404, Z -7.1667, A 0.000, B 0.000, C 0.000 }
gfCNCPoint5[8148] = {X 515.0460, Y 70.4852, Z -7.1667, A 0.000, B 0.000, C 0.000 }
gfCNCPoint5[8149] = {X 512.7278, Y 69.8972, Z -7.1667, A 0.000, B 0.000, C 0.000 }
gfCNCPoint5[8150] = {X 510.4794, Y 69.0822, Z -7.1667, A 0.000, B 0.000, C 0.000 }
gfCNCPoint5[8151] = {X 509.6267, Y 68.7047, Z -7.1667, A 0.000, B 0.000, C 0.000 }
gfCNCPoint5[8152] = {X 508.7892, Y 68.2944, Z -7.1667, A 0.000, B 0.000, C 0.000 }
gfCNCPoint5[8153] = {X 507.1697, Y 68.6594, Z -7.1667, A 0.000, B 0.000, C 0.000 }
gfCNCPoint5[8154] = {X 505.5289, Y 68.9119, Z -7.1667, A 0.000, B 0.000, C 0.000 }
gfCNCPoint5[8155] = {X 504.1112, Y 69.0379, Z -7.1667, A 0.000, B 0.000, C 0.000 }
gfCNCPoint5[8156] = {X 502.6885, Y 69.0800, Z -7.1667, A 0.000, B 0.000, C 0.000 }
gfCNCPoint5[8157] = {X 502.0391, Y 69.0800, Z -7.1667, A 0.000, B 0.000, C 0.000 }
gfCNCPoint5[8158] = {X 501.1778, Y 71.1315, Z -7.1667, A 0.000, B 0.000, C 0.000 }
gfCNCPoint5[8159] = {X 500.1611, Y 73.1105, Z -7.1667, A 0.000, B 0.000, C 0.000 }
gfCNCPoint5[8160] = {X 500.1611, Y 73.6951, Z -7.1667, A 0.000, B 0.000, C 0.000 }
gfCNCPoint5[8161] = {X 507.6812, Y 73.6951, Z -7.1667, A 0.000, B 0.000, C 0.000 }
gfCNCPoint5[8162] = {X 507.6812, Y 76.0951, Z -7.1667, A 0.000, B 0.000, C 0.000 }
gfCNCPoint5[8163] = {X 576.0967, Y 76.0951, Z -7.1667, A 0.000, B 0.000, C 0.000 }
gfCNCPoint5[8164] = {X 576.0967, Y 72.8901, Z -7.1667, A 0.000, B 0.000, C 0.000 }
gfCNCPoint5[8165] = {X 575.7179, Y 72.8147, Z -7.1667, A 0.000, B 0.000, C 0.000 }
gfCNCPoint5[8166] = {X 575.3401, Y 72.7341, Z -7.1667, A 0.000, B 0.000, C 0.000 }
gfCNCPoint5[8167] = {X 573.3201, Y 73.1034, Z -7.1667, A 0.000, B 0.000, C 0.000 }
gfCNCPoint5[8168] = {X 571.2786, Y 73.3258, Z -7.1667, A 0.000, B 0.000, C 0.000 }
gfCNCPoint5[8169] = {X 569.2264, Y 73.4000, Z -7.1667, A 0.000, B 0.000, C 0.000 }
gfCNCPoint5[8170] = {X 562.4443, Y 73.4000, Z -7.1667, A 0.000, B 0.000, C 0.000 }
gfCNCPoint5[8171] = {X 560.3342, Y 73.3215, Z -7.1667, A 0.000, B 0.000, C 0.000 }
gfCNCPoint5[8172] = {X 558.2357, Y 73.0864, Z -7.1667, A 0.000, B 0.000, C 0.000 }
gfCNCPoint5[8173] = {X 556.1606, Y 72.6961, Z -7.1667, A 0.000, B 0.000, C 0.000 }
gfCNCPoint5[8174] = {X 554.1201, Y 72.1527, Z -7.1667, A 0.000, B 0.000, C 0.000 }
gfCNCPoint5[8175] = {X 552.1257, Y 71.4592, Z -7.1667, A 0.000, B 0.000, C 0.000 }
gfCNCPoint5[8176] = {X 549.9767, Y 70.5171, Z -7.1667, A 0.000, B 0.000, C 0.000 }
gfCNCPoint5[8177] = {X 547.9129, Y 69.4008, Z -7.1667, A 0.000, B 0.000, C 0.000 }
gfCNCPoint5[8178] = {X 545.9482, Y 68.1179, Z -7.1667, A 0.000, B 0.000, C 0.000 }
gfCNCPoint5[8179] = {X 544.0962, Y 66.6773, Z -7.1667, A 0.000, B 0.000, C 0.000 }
gfCNCPoint5[8180] = {X 543.8506, Y 66.6785, Z -7.1667, A 0.000, B 0.000, C 0.000 }
gfCNCPoint5[8181] = {X 543.6050, Y 66.6769, Z -7.1667, A 0.000, B 0.000, C 0.000 }
gfCNCPoint5[8182] = {X 529.2671, Y 66.6772, Z -7.1667, A 0.000, B 0.000, C 0.000 }
gfCNCPoint5[8183] = {X 527.1798, Y 67.4797, Z -7.1667, A 0.000, B 0.000, C 0.000 }
gfCNCPoint5[8184] = {X 525.0214, Y 68.0645, Z -7.1667, A 0.000, B 0.000, C 0.000 }
gfCNCPoint5[8185] = {X 522.8146, Y 68.4255, Z -7.1667, A 0.000, B 0.000, C 0.000 }
gfCNCPoint5[8186] = {X 520.5823, Y 68.5589, Z -7.1667, A 0.000, B 0.000, C 0.000 }
gfCNCPoint5[8187] = {X 519.7998, Y 68.5591, Z -7.1667, A 0.000, B 0.000, C 0.000 }
gfCNCPoint5[8188] = {X 517.5593, Y 68.4430, Z -7.1667, A 0.000, B 0.000, C 0.000 }
gfCNCPoint5[8189] = {X 515.3429, Y 68.0961, Z -7.1667, A 0.000, B 0.000, C 0.000 }
gfCNCPoint5[8190] = {X 513.1742, Y 67.5219, Z -7.1667, A 0.000, B 0.000, C 0.000 }
gfCNCPoint5[8191] = {X 511.0764, Y 66.7267, Z -7.1667, A 0.000, B 0.000, C 0.000 }
gfCNCPoint5[8192] = {X 509.0720, Y 65.7189, Z -7.1667, A 0.000, B 0.000, C 0.000 }
gfCNCPoint5[8193] = {X 506.9797, Y 66.2511, Z -7.1667, A 0.000, B 0.000, C 0.000 }
gfCNCPoint5[8194] = {X 504.8448, Y 66.5725, Z -7.1667, A 0.000, B 0.000, C 0.000 }
gfCNCPoint5[8195] = {X 502.6885, Y 66.6800, Z -7.1667, A 0.000, B 0.000, C 0.000 }
gfCNCPoint5[8196] = {X 500.3217, Y 66.6800, Z -7.1667, A 0.000, B 0.000, C 0.000 }
gfCNCPoint5[8197] = {X 499.6233, Y 68.6749, Z -7.1667, A 0.000, B 0.000, C 0.000 }
gfCNCPoint5[8198] = {X 498.7679, Y 70.6078, Z -7.1667, A 0.000, B 0.000, C 0.000 }
gfCNCPoint5[8199] = {X 497.7611, Y 72.4663, Z -7.1667, A 0.000, B 0.000, C 0.000 }
gfCNCPoint5[8200] = {X 497.7612, Y 76.0951, Z -7.1667, A 0.000, B 0.000, C 0.000 }
gfCNCPoint5[8201] = {X 507.6812, Y 76.0951, Z -7.1667, A 0.000, B 0.000, C 0.000 }
gfCNCPoint5[8202] = {X 507.6812, Y 78.4951, Z -7.1667, A 0.000, B 0.000, C 0.000 }
gfCNCPoint5[8203] = {X 578.4967, Y 78.4951, Z -7.1667, A 0.000, B 0.000, C 0.000 }
gfCNCPoint5[8204] = {X 578.4967, Y 70.8313, Z -7.1667, A 0.000, B 0.000, C 0.000 }
gfCNCPoint5[8205] = {X 576.9098, Y 70.5998, Z -7.1667, A 0.000, B 0.000, C 0.000 }
gfCNCPoint5[8206] = {X 575.3401, Y 70.2710, Z -7.1667, A 0.000, B 0.000, C 0.000 }
gfCNCPoint5[8207] = {X 573.3236, Y 70.6751, Z -7.1667, A 0.000, B 0.000, C 0.000 }
gfCNCPoint5[8208] = {X 571.2815, Y 70.9187, Z -7.1667, A 0.000, B 0.000, C 0.000 }
gfCNCPoint5[8209] = {X 569.2264, Y 71.0000, Z -7.1667, A 0.000, B 0.000, C 0.000 }
gfCNCPoint5[8210] = {X 562.4443, Y 71.0000, Z -7.1667, A 0.000, B 0.000, C 0.000 }
gfCNCPoint5[8211] = {X 560.0514, Y 70.8897, Z -7.1667, A 0.000, B 0.000, C 0.000 }
gfCNCPoint5[8212] = {X 557.6789, Y 70.5595, Z -7.1667, A 0.000, B 0.000, C 0.000 }
gfCNCPoint5[8213] = {X 555.3468, Y 70.0125, Z -7.1667, A 0.000, B 0.000, C 0.000 }
gfCNCPoint5[8214] = {X 553.0749, Y 69.2531, Z -7.1667, A 0.000, B 0.000, C 0.000 }
gfCNCPoint5[8215] = {X 550.8826, Y 68.2879, Z -7.1667, A 0.000, B 0.000, C 0.000 }
gfCNCPoint5[8216] = {X 548.7884, Y 67.1250, Z -7.1667, A 0.000, B 0.000, C 0.000 }
gfCNCPoint5[8217] = {X 546.8101, Y 65.7743, Z -7.1667, A 0.000, B 0.000, C 0.000 }
gfCNCPoint5[8218] = {X 544.9645, Y 64.2473, Z -7.1667, A 0.000, B 0.000, C 0.000 }
gfCNCPoint5[8219] = {X 544.2925, Y 64.2738, Z -7.1667, A 0.000, B 0.000, C 0.000 }
gfCNCPoint5[8220] = {X 543.6199, Y 64.2769, Z -7.1667, A 0.000, B 0.000, C 0.000 }
gfCNCPoint5[8221] = {X 528.7422, Y 64.2772, Z -7.1667, A 0.000, B 0.000, C 0.000 }
gfCNCPoint5[8222] = {X 526.7885, Y 65.0789, Z -7.1667, A 0.000, B 0.000, C 0.000 }
gfCNCPoint5[8223] = {X 524.7594, Y 65.6639, Z -7.1667, A 0.000, B 0.000, C 0.000 }
gfCNCPoint5[8224] = {X 522.6788, Y 66.0253, Z -7.1667, A 0.000, B 0.000, C 0.000 }
gfCNCPoint5[8225] = {X 520.5712, Y 66.1589, Z -7.1667, A 0.000, B 0.000, C 0.000 }
gfCNCPoint5[8226] = {X 519.7998, Y 66.1591, Z -7.1667, A 0.000, B 0.000, C 0.000 }
gfCNCPoint5[8227] = {X 517.9641, Y 66.0715, Z -7.1667, A 0.000, B 0.000, C 0.000 }
gfCNCPoint5[8228] = {X 516.1450, Y 65.8096, Z -7.1667, A 0.000, B 0.000, C 0.000 }
gfCNCPoint5[8229] = {X 514.3592, Y 65.3756, Z -7.1667, A 0.000, B 0.000, C 0.000 }
gfCNCPoint5[8230] = {X 512.6228, Y 64.7735, Z -7.1667, A 0.000, B 0.000, C 0.000 }
gfCNCPoint5[8231] = {X 510.9516, Y 64.0089, Z -7.1667, A 0.000, B 0.000, C 0.000 }
gfCNCPoint5[8232] = {X 509.3609, Y 63.0886, Z -7.1667, A 0.000, B 0.000, C 0.000 }
gfCNCPoint5[8233] = {X 507.7389, Y 63.6068, Z -7.1667, A 0.000, B 0.000, C 0.000 }
gfCNCPoint5[8234] = {X 506.0774, Y 63.9798, Z -7.1667, A 0.000, B 0.000, C 0.000 }
gfCNCPoint5[8235] = {X 504.3896, Y 64.2048, Z -7.1667, A 0.000, B 0.000, C 0.000 }
gfCNCPoint5[8236] = {X 502.6885, Y 64.2800, Z -7.1667, A 0.000, B 0.000, C 0.000 }
gfCNCPoint5[8237] = {X 498.4791, Y 64.2800, Z -7.1667, A 0.000, B 0.000, C 0.000 }
gfCNCPoint5[8238] = {X 497.9417, Y 66.2500, Z -7.1667, A 0.000, B 0.000, C 0.000 }
gfCNCPoint5[8239] = {X 497.2394, Y 68.1675, Z -7.1667, A 0.000, B 0.000, C 0.000 }
gfCNCPoint5[8240] = {X 496.3771, Y 70.0185, Z -7.1667, A 0.000, B 0.000, C 0.000 }
gfCNCPoint5[8241] = {X 495.3611, Y 71.7899, Z -7.1667, A 0.000, B 0.000, C 0.000 }
gfCNCPoint5[8242] = {X 495.3612, Y 78.4951, Z -7.1667, A 0.000, B 0.000, C 0.000 }
gfCNCPoint5[8243] = {X 507.6812, Y 78.4951, Z -7.1667, A 0.000, B 0.000, C 0.000 }
gfCNCPoint5[8244] = {X 507.6812, Y 80.8951, Z -7.1667, A 0.000, B 0.000, C 0.000 }
gfCNCPoint5[8245] = {X 580.8967, Y 80.8951, Z -7.1667, A 0.000, B 0.000, C 0.000 }
gfCNCPoint5[8246] = {X 580.8967, Y 68.5934, Z -7.1667, A 0.000, B 0.000, C 0.000 }
gfCNCPoint5[8247] = {X 579.0253, Y 68.4747, Z -7.1667, A 0.000, B 0.000, C 0.000 }
gfCNCPoint5[8248] = {X 577.1692, Y 68.2078, Z -7.1667, A 0.000, B 0.000, C 0.000 }
gfCNCPoint5[8249] = {X 575.3401, Y 67.7943, Z -7.1667, A 0.000, B 0.000, C 0.000 }
gfCNCPoint5[8250] = {X 573.3283, Y 68.2408, Z -7.1667, A 0.000, B 0.000, C 0.000 }
gfCNCPoint5[8251] = {X 571.2852, Y 68.5100, Z -7.1667, A 0.000, B 0.000, C 0.000 }
gfCNCPoint5[8252] = {X 569.2264, Y 68.6000, Z -7.1667, A 0.000, B 0.000, C 0.000 }
gfCNCPoint5[8253] = {X 562.4443, Y 68.6000, Z -7.1667, A 0.000, B 0.000, C 0.000 }
gfCNCPoint5[8254] = {X 560.1445, Y 68.4877, Z -7.1667, A 0.000, B 0.000, C 0.000 }
gfCNCPoint5[8255] = {X 557.8666, Y 68.1518, Z -7.1667, A 0.000, B 0.000, C 0.000 }
gfCNCPoint5[8256] = {X 555.6322, Y 67.5955, Z -7.1667, A 0.000, B 0.000, C 0.000 }
gfCNCPoint5[8257] = {X 553.4627, Y 66.8241, Z -7.1667, A 0.000, B 0.000, C 0.000 }
gfCNCPoint5[8258] = {X 551.3787, Y 65.8450, Z -7.1667, A 0.000, B 0.000, C 0.000 }
gfCNCPoint5[8259] = {X 549.4001, Y 64.6674, Z -7.1667, A 0.000, B 0.000, C 0.000 }
gfCNCPoint5[8260] = {X 547.5456, Y 63.3027, Z -7.1667, A 0.000, B 0.000, C 0.000 }
gfCNCPoint5[8261] = {X 545.8329, Y 61.7637, Z -7.1667, A 0.000, B 0.000, C 0.000 }
gfCNCPoint5[8262] = {X 544.7362, Y 61.8561, Z -7.1667, A 0.000, B 0.000, C 0.000 }
gfCNCPoint5[8263] = {X 543.6358, Y 61.8769, Z -7.1667, A 0.000, B 0.000, C 0.000 }
gfCNCPoint5[8264] = {X 528.1819, Y 61.8772, Z -7.1667, A 0.000, B 0.000, C 0.000 }
gfCNCPoint5[8265] = {X 526.3716, Y 62.6779, Z -7.1667, A 0.000, B 0.000, C 0.000 }
gfCNCPoint5[8266] = {X 524.4806, Y 63.2631, Z -7.1667, A 0.000, B 0.000, C 0.000 }
gfCNCPoint5[8267] = {X 522.5344, Y 63.6251, Z -7.1667, A 0.000, B 0.000, C 0.000 }
gfCNCPoint5[8268] = {X 520.5594, Y 63.7589, Z -7.1667, A 0.000, B 0.000, C 0.000 }
gfCNCPoint5[8269] = {X 519.7998, Y 63.7591, Z -7.1667, A 0.000, B 0.000, C 0.000 }
gfCNCPoint5[8270] = {X 517.9902, Y 63.6618, Z -7.1667, A 0.000, B 0.000, C 0.000 }
gfCNCPoint5[8271] = {X 516.2015, Y 63.3711, Z -7.1667, A 0.000, B 0.000, C 0.000 }
gfCNCPoint5[8272] = {X 514.4543, Y 62.8904, Z -7.1667, A 0.000, B 0.000, C 0.000 }
gfCNCPoint5[8273] = {X 512.7687, Y 62.2251, Z -7.1667, A 0.000, B 0.000, C 0.000 }
gfCNCPoint5[8274] = {X 511.1641, Y 61.3829, Z -7.1667, A 0.000, B 0.000, C 0.000 }
gfCNCPoint5[8275] = {X 509.6590, Y 60.3735, Z -7.1667, A 0.000, B 0.000, C 0.000 }
gfCNCPoint5[8276] = {X 507.9866, Y 61.0270, Z -7.1667, A 0.000, B 0.000, C 0.000 }
gfCNCPoint5[8277] = {X 506.2542, Y 61.4991, Z -7.1667, A 0.000, B 0.000, C 0.000 }
gfCNCPoint5[8278] = {X 504.4815, Y 61.7845, Z -7.1667, A 0.000, B 0.000, C 0.000 }
gfCNCPoint5[8279] = {X 502.6885, Y 61.8800, Z -7.1667, A 0.000, B 0.000, C 0.000 }
gfCNCPoint5[8280] = {X 496.4789, Y 61.8800, Z -7.1667, A 0.000, B 0.000, C 0.000 }
gfCNCPoint5[8281] = {X 496.1193, Y 63.8329, Z -7.1667, A 0.000, B 0.000, C 0.000 }
gfCNCPoint5[8282] = {X 495.5824, Y 65.7448, Z -7.1667, A 0.000, B 0.000, C 0.000 }
gfCNCPoint5[8283] = {X 494.8729, Y 67.5994, Z -7.1667, A 0.000, B 0.000, C 0.000 }
gfCNCPoint5[8284] = {X 493.9967, Y 69.3814, Z -7.1667, A 0.000, B 0.000, C 0.000 }
gfCNCPoint5[8285] = {X 492.9611, Y 71.0758, Z -7.1667, A 0.000, B 0.000, C 0.000 }
gfCNCPoint5[8286] = {X 492.9613, Y 80.8951, Z -7.1667, A 0.000, B 0.000, C 0.000 }
gfCNCPoint5[8287] = {X 507.6812, Y 80.8951, Z -7.1667, A 0.000, B 0.000, C 0.000 }
gfCNCPoint5[8288] = {X 507.6812, Y 83.2951, Z -7.1667, A 0.000, B 0.000, C 0.000 }
gfCNCPoint5[8289] = {X 583.2967, Y 83.2951, Z -7.1667, A 0.000, B 0.000, C 0.000 }
gfCNCPoint5[8290] = {X 583.2967, Y 66.1198, Z -7.1667, A 0.000, B 0.000, C 0.000 }
gfCNCPoint5[8291] = {X 581.2873, Y 66.1993, Z -7.1667, A 0.000, B 0.000, C 0.000 }
gfCNCPoint5[8292] = {X 579.2794, Y 66.0882, Z -7.1667, A 0.000, B 0.000, C 0.000 }
gfCNCPoint5[8293] = {X 577.2910, Y 65.7873, Z -7.1667, A 0.000, B 0.000, C 0.000 }
gfCNCPoint5[8294] = {X 575.3401, Y 65.2993, Z -7.1667, A 0.000, B 0.000, C 0.000 }
gfCNCPoint5[8295] = {X 573.3348, Y 65.7981, Z -7.1667, A 0.000, B 0.000, C 0.000 }
gfCNCPoint5[8296] = {X 571.2904, Y 66.0993, Z -7.1667, A 0.000, B 0.000, C 0.000 }
gfCNCPoint5[8297] = {X 569.2264, Y 66.2000, Z -7.1667, A 0.000, B 0.000, C 0.000 }
gfCNCPoint5[8298] = {X 562.4443, Y 66.2000, Z -7.1667, A 0.000, B 0.000, C 0.000 }
gfCNCPoint5[8299] = {X 560.3663, Y 66.0979, Z -7.1667, A 0.000, B 0.000, C 0.000 }
gfCNCPoint5[8300] = {X 558.3084, Y 65.7926, Z -7.1667, A 0.000, B 0.000, C 0.000 }
gfCNCPoint5[8301] = {X 556.2903, Y 65.2871, Z -7.1667, A 0.000, B 0.000, C 0.000 }
gfCNCPoint5[8302] = {X 554.3314, Y 64.5862, Z -7.1667, A 0.000, B 0.000, C 0.000 }
gfCNCPoint5[8303] = {X 552.4507, Y 63.6967, Z -7.1667, A 0.000, B 0.000, C 0.000 }
gfCNCPoint5[8304] = {X 550.6662, Y 62.6272, Z -7.1667, A 0.000, B 0.000, C 0.000 }
gfCNCPoint5[8305] = {X 548.9952, Y 61.3878, Z -7.1667, A 0.000, B 0.000, C 0.000 }
gfCNCPoint5[8306] = {X 547.4536, Y 59.9907, Z -7.1667, A 0.000, B 0.000, C 0.000 }
gfCNCPoint5[8307] = {X 547.0724, Y 59.5994, Z -7.1667, A 0.000, B 0.000, C 0.000 }
gfCNCPoint5[8308] = {X 546.7013, Y 59.1985, Z -7.1667, A 0.000, B 0.000, C 0.000 }
gfCNCPoint5[8309] = {X 545.1844, Y 59.4185, Z -7.1667, A 0.000, B 0.000, C 0.000 }
gfCNCPoint5[8310] = {X 543.6528, Y 59.4769, Z -7.1667, A 0.000, B 0.000, C 0.000 }
gfCNCPoint5[8311] = {X 527.5781, Y 59.4772, Z -7.1667, A 0.000, B 0.000, C 0.000 }
gfCNCPoint5[8312] = {X 525.9209, Y 60.2775, Z -7.1667, A 0.000, B 0.000, C 0.000 }
gfCNCPoint5[8313] = {X 524.1764, Y 60.8634, Z -7.1667, A 0.000, B 0.000, C 0.000 }
gfCNCPoint5[8314] = {X 522.3721, Y 61.2259, Z -7.1667, A 0.000, B 0.000, C 0.000 }
gfCNCPoint5[8315] = {X 520.5366, Y 61.3590, Z -7.1667, A 0.000, B 0.000, C 0.000 }
gfCNCPoint5[8316] = {X 519.7998, Y 61.3591, Z -7.1667, A 0.000, B 0.000, C 0.000 }
gfCNCPoint5[8317] = {X 518.0043, Y 61.2474, Z -7.1667, A 0.000, B 0.000, C 0.000 }
gfCNCPoint5[8318] = {X 516.2365, Y 60.9138, Z -7.1667, A 0.000, B 0.000, C 0.000 }
gfCNCPoint5[8319] = {X 514.5237, Y 60.3637, Z -7.1667, A 0.000, B 0.000, C 0.000 }
gfCNCPoint5[8320] = {X 512.8923, Y 59.6054, Z -7.1667, A 0.000, B 0.000, C 0.000 }
gfCNCPoint5[8321] = {X 511.3676, Y 58.6507, Z -7.1667, A 0.000, B 0.000, C 0.000 }
gfCNCPoint5[8322] = {X 509.9730, Y 57.5142, Z -7.1667, A 0.000, B 0.000, C 0.000 }
gfCNCPoint5[8323] = {X 508.6156, Y 58.2113, Z -7.1667, A 0.000, B 0.000, C 0.000 }
gfCNCPoint5[8324] = {X 507.1924, Y 58.7617, Z -7.1667, A 0.000, B 0.000, C 0.000 }
gfCNCPoint5[8325] = {X 505.7192, Y 59.1593, Z -7.1667, A 0.000, B 0.000, C 0.000 }
gfCNCPoint5[8326] = {X 504.2123, Y 59.3996, Z -7.1667, A 0.000, B 0.000, C 0.000 }
gfCNCPoint5[8327] = {X 502.6885, Y 59.4800, Z -7.1667, A 0.000, B 0.000, C 0.000 }
gfCNCPoint5[8328] = {X 496.2450, Y 59.4800, Z -7.1667, A 0.000, B 0.000, C 0.000 }
gfCNCPoint5[8329] = {X 495.2580, Y 59.4463, Z -7.1667, A 0.000, B 0.000, C 0.000 }
gfCNCPoint5[8330] = {X 494.2756, Y 59.3454, Z -7.1667, A 0.000, B 0.000, C 0.000 }
gfCNCPoint5[8331] = {X 494.1342, Y 61.3003, Z -7.1667, A 0.000, B 0.000, C 0.000 }
gfCNCPoint5[8332] = {X 493.7951, Y 63.2307, Z -7.1667, A 0.000, B 0.000, C 0.000 }
gfCNCPoint5[8333] = {X 493.2618, Y 65.1168, Z -7.1667, A 0.000, B 0.000, C 0.000 }
gfCNCPoint5[8334] = {X 492.5397, Y 66.9389, Z -7.1667, A 0.000, B 0.000, C 0.000 }
gfCNCPoint5[8335] = {X 491.6364, Y 68.6783, Z -7.1667, A 0.000, B 0.000, C 0.000 }
gfCNCPoint5[8336] = {X 490.5611, Y 70.3170, Z -7.1667, A 0.000, B 0.000, C 0.000 }
gfCNCPoint5[8337] = {X 490.5613, Y 83.2951, Z -7.1667, A 0.000, B 0.000, C 0.000 }
gfCNCPoint5[8338] = {X 507.6812, Y 83.2951, Z -7.1667, A 0.000, B 0.000, C 0.000 }
gfCNCPoint5[8339] = {X 507.6812, Y 85.6951, Z -7.1667, A 0.000, B 0.000, C 0.000 }
gfCNCPoint5[8340] = {X 585.6967, Y 85.6951, Z -7.1667, A 0.000, B 0.000, C 0.000 }
gfCNCPoint5[8341] = {X 585.6967, Y 63.3150, Z -7.1667, A 0.000, B 0.000, C 0.000 }
gfCNCPoint5[8342] = {X 584.3996, Y 63.5678, Z -7.1667, A 0.000, B 0.000, C 0.000 }
gfCNCPoint5[8343] = {X 583.0880, Y 63.7288, Z -7.1667, A 0.000, B 0.000, C 0.000 }
gfCNCPoint5[8344] = {X 581.1243, Y 63.7971, Z -7.1667, A 0.000, B 0.000, C 0.000 }
gfCNCPoint5[8345] = {X 579.1642, Y 63.6600, Z -7.1667, A 0.000, B 0.000, C 0.000 }
gfCNCPoint5[8346] = {X 577.2291, Y 63.3192, Z -7.1667, A 0.000, B 0.000, C 0.000 }
gfCNCPoint5[8347] = {X 575.3401, Y 62.7781, Z -7.1667, A 0.000, B 0.000, C 0.000 }
gfCNCPoint5[8348] = {X 573.3441, Y 63.3435, Z -7.1667, A 0.000, B 0.000, C 0.000 }
gfCNCPoint5[8349] = {X 571.2979, Y 63.6855, Z -7.1667, A 0.000, B 0.000, C 0.000 }
gfCNCPoint5[8350] = {X 569.2264, Y 63.8000, Z -7.1667, A 0.000, B 0.000, C 0.000 }
gfCNCPoint5[8351] = {X 562.4443, Y 63.8000, Z -7.1667, A 0.000, B 0.000, C 0.000 }
gfCNCPoint5[8352] = {X 560.3394, Y 63.6818, Z -7.1667, A 0.000, B 0.000, C 0.000 }
gfCNCPoint5[8353] = {X 558.2609, Y 63.3286, Z -7.1667, A 0.000, B 0.000, C 0.000 }
gfCNCPoint5[8354] = {X 556.2351, Y 62.7450, Z -7.1667, A 0.000, B 0.000, C 0.000 }
gfCNCPoint5[8355] = {X 554.2873, Y 61.9382, Z -7.1667, A 0.000, B 0.000, C 0.000 }
gfCNCPoint5[8356] = {X 552.4421, Y 60.9184, Z -7.1667, A 0.000, B 0.000, C 0.000 }
gfCNCPoint5[8357] = {X 550.7227, Y 59.6984, Z -7.1667, A 0.000, B 0.000, C 0.000 }
gfCNCPoint5[8358] = {X 549.1507, Y 58.2936, Z -7.1667, A 0.000, B 0.000, C 0.000 }
gfCNCPoint5[8359] = {X 548.3316, Y 57.4206, Z -7.1667, A 0.000, B 0.000, C 0.000 }
gfCNCPoint5[8360] = {X 547.5697, Y 56.4973, Z -7.1667, A 0.000, B 0.000, C 0.000 }
gfCNCPoint5[8361] = {X 546.2940, Y 56.8323, Z -7.1667, A 0.000, B 0.000, C 0.000 }
gfCNCPoint5[8362] = {X 544.9894, Y 57.0263, Z -7.1667, A 0.000, B 0.000, C 0.000 }
gfCNCPoint5[8363] = {X 543.6714, Y 57.0769, Z -7.1667, A 0.000, B 0.000, C 0.000 }
gfCNCPoint5[8364] = {X 526.9186, Y 57.0772, Z -7.1667, A 0.000, B 0.000, C 0.000 }
gfCNCPoint5[8365] = {X 525.4331, Y 57.8755, Z -7.1667, A 0.000, B 0.000, C 0.000 }
gfCNCPoint5[8366] = {X 523.8519, Y 58.4619, Z -7.1667, A 0.000, B 0.000, C 0.000 }
gfCNCPoint5[8367] = {X 522.2051, Y 58.8254, Z -7.1667, A 0.000, B 0.000, C 0.000 }
gfCNCPoint5[8368] = {X 520.5240, Y 58.9590, Z -7.1667, A 0.000, B 0.000, C 0.000 }
gfCNCPoint5[8369] = {X 519.7998, Y 58.9591, Z -7.1667, A 0.000, B 0.000, C 0.000 }
gfCNCPoint5[8370] = {X 518.2467, Y 58.8589, Z -7.1667, A 0.000, B 0.000, C 0.000 }
gfCNCPoint5[8371] = {X 516.7195, Y 58.5598, Z -7.1667, A 0.000, B 0.000, C 0.000 }
gfCNCPoint5[8372] = {X 515.2433, Y 58.0668, Z -7.1667, A 0.000, B 0.000, C 0.000 }
gfCNCPoint5[8373] = {X 513.8428, Y 57.3882, Z -7.1667, A 0.000, B 0.000, C 0.000 }
gfCNCPoint5[8374] = {X 512.5411, Y 56.5351, Z -7.1667, A 0.000, B 0.000, C 0.000 }
gfCNCPoint5[8375] = {X 511.3600, Y 55.5218, Z -7.1667, A 0.000, B 0.000, C 0.000 }
gfCNCPoint5[8376] = {X 510.3189, Y 54.3650, Z -7.1667, A 0.000, B 0.000, C 0.000 }
gfCNCPoint5[8377] = {X 508.9711, Y 55.3177, Z -7.1667, A 0.000, B 0.000, C 0.000 }
gfCNCPoint5[8378] = {X 507.5060, Y 56.0778, Z -7.1667, A 0.000, B 0.000, C 0.000 }
gfCNCPoint5[8379] = {X 505.9510, Y 56.6311, Z -7.1667, A 0.000, B 0.000, C 0.000 }
gfCNCPoint5[8380] = {X 504.3351, Y 56.9672, Z -7.1667, A 0.000, B 0.000, C 0.000 }
gfCNCPoint5[8381] = {X 502.6885, Y 57.0800, Z -7.1667, A 0.000, B 0.000, C 0.000 }
gfCNCPoint5[8382] = {X 496.2450, Y 57.0800, Z -7.1667, A 0.000, B 0.000, C 0.000 }
gfCNCPoint5[8383] = {X 495.4216, Y 57.0519, Z -7.1667, A 0.000, B 0.000, C 0.000 }
gfCNCPoint5[8384] = {X 494.6020, Y 56.9677, Z -7.1667, A 0.000, B 0.000, C 0.000 }
gfCNCPoint5[8385] = {X 493.1719, Y 56.6826, Z -7.1667, A 0.000, B 0.000, C 0.000 }
gfCNCPoint5[8386] = {X 491.7866, Y 56.2272, Z -7.1667, A 0.000, B 0.000, C 0.000 }
gfCNCPoint5[8387] = {X 491.8566, Y 57.1124, Z -7.1667, A 0.000, B 0.000, C 0.000 }
gfCNCPoint5[8388] = {X 491.8800, Y 58.0000, Z -7.1667, A 0.000, B 0.000, C 0.000 }
gfCNCPoint5[8389] = {X 491.8794, Y 59.0735, Z -7.1667, A 0.000, B 0.000, C 0.000 }
gfCNCPoint5[8390] = {X 491.8781, Y 59.1839, Z -7.1667, A 0.000, B 0.000, C 0.000 }
gfCNCPoint5[8391] = {X 491.8762, Y 59.2942, Z -7.1667, A 0.000, B 0.000, C 0.000 }
gfCNCPoint5[8392] = {X 491.7363, Y 61.1316, Z -7.1667, A 0.000, B 0.000, C 0.000 }
gfCNCPoint5[8393] = {X 491.3971, Y 62.9427, Z -7.1667, A 0.000, B 0.000, C 0.000 }
gfCNCPoint5[8394] = {X 490.8625, Y 64.7061, Z -7.1667, A 0.000, B 0.000, C 0.000 }
gfCNCPoint5[8395] = {X 490.1388, Y 66.4007, Z -7.1667, A 0.000, B 0.000, C 0.000 }
gfCNCPoint5[8396] = {X 489.2348, Y 68.0063, Z -7.1667, A 0.000, B 0.000, C 0.000 }
gfCNCPoint5[8397] = {X 488.1611, Y 69.5038, Z -7.1667, A 0.000, B 0.000, C 0.000 }
gfCNCPoint5[8398] = {X 488.1613, Y 85.6951, Z -7.1667, A 0.000, B 0.000, C 0.000 }
gfCNCPoint5[8399] = {X 507.6812, Y 85.6951, Z -7.1667, A 0.000, B 0.000, C 0.000 }
gfCNCPoint5[8400] = {X 507.6812, Y 88.0951, Z -7.1667, A 0.000, B 0.000, C 0.000 }
gfCNCPoint5[8401] = {X 588.0967, Y 88.0951, Z -7.1667, A 0.000, B 0.000, C 0.000 }
gfCNCPoint5[8402] = {X 588.0967, Y 60.4645, Z -7.1667, A 0.000, B 0.000, C 0.000 }
gfCNCPoint5[8403] = {X 587.7999, Y 60.3565, Z -7.1667, A 0.000, B 0.000, C 0.000 }
gfCNCPoint5[8404] = {X 587.5052, Y 60.2427, Z -7.1667, A 0.000, B 0.000, C 0.000 }
gfCNCPoint5[8405] = {X 586.3439, Y 60.6540, Z -7.1667, A 0.000, B 0.000, C 0.000 }
gfCNCPoint5[8406] = {X 585.1550, Y 60.9769, Z -7.1667, A 0.000, B 0.000, C 0.000 }
gfCNCPoint5[8407] = {X 583.5153, Y 61.2699, Z -7.1667, A 0.000, B 0.000, C 0.000 }
gfCNCPoint5[8408] = {X 581.8544, Y 61.3951, Z -7.1667, A 0.000, B 0.000, C 0.000 }
gfCNCPoint5[8409] = {X 580.1893, Y 61.3512, Z -7.1667, A 0.000, B 0.000, C 0.000 }
gfCNCPoint5[8410] = {X 578.5372, Y 61.1386, Z -7.1667, A 0.000, B 0.000, C 0.000 }
gfCNCPoint5[8411] = {X 576.9153, Y 60.7595, Z -7.1667, A 0.000, B 0.000, C 0.000 }
gfCNCPoint5[8412] = {X 575.3401, Y 60.2178, Z -7.1667, A 0.000, B 0.000, C 0.000 }
gfCNCPoint5[8413] = {X 573.8611, Y 60.7315, Z -7.1667, A 0.000, B 0.000, C 0.000 }
gfCNCPoint5[8414] = {X 572.3399, Y 61.1017, Z -7.1667, A 0.000, B 0.000, C 0.000 }
gfCNCPoint5[8415] = {X 570.7903, Y 61.3253, Z -7.1667, A 0.000, B 0.000, C 0.000 }
gfCNCPoint5[8416] = {X 569.2264, Y 61.4000, Z -7.1667, A 0.000, B 0.000, C 0.000 }
gfCNCPoint5[8417] = {X 562.4443, Y 61.4000, Z -7.1667, A 0.000, B 0.000, C 0.000 }
gfCNCPoint5[8418] = {X 560.6081, Y 61.2969, Z -7.1667, A 0.000, B 0.000, C 0.000 }
gfCNCPoint5[8419] = {X 558.7950, Y 60.9888, Z -7.1667, A 0.000, B 0.000, C 0.000 }
gfCNCPoint5[8420] = {X 557.0277, Y 60.4797, Z -7.1667, A 0.000, B 0.000, C 0.000 }
gfCNCPoint5[8421] = {X 555.3286, Y 59.7759, Z -7.1667, A 0.000, B 0.000, C 0.000 }
gfCNCPoint5[8422] = {X 553.7190, Y 58.8863, Z -7.1667, A 0.000, B 0.000, C 0.000 }
gfCNCPoint5[8423] = {X 552.2191, Y 57.8220, Z -7.1667, A 0.000, B 0.000, C 0.000 }
gfCNCPoint5[8424] = {X 550.8478, Y 56.5966, Z -7.1667, A 0.000, B 0.000, C 0.000 }
gfCNCPoint5[8425] = {X 549.5516, Y 55.1360, Z -7.1667, A 0.000, B 0.000, C 0.000 }
gfCNCPoint5[8426] = {X 548.4383, Y 53.5317, Z -7.1667, A 0.000, B 0.000, C 0.000 }
gfCNCPoint5[8427] = {X 547.3163, Y 54.0434, Z -7.1667, A 0.000, B 0.000, C 0.000 }
gfCNCPoint5[8428] = {X 546.1384, Y 54.4084, Z -7.1667, A 0.000, B 0.000, C 0.000 }
gfCNCPoint5[8429] = {X 544.9237, Y 54.6207, Z -7.1667, A 0.000, B 0.000, C 0.000 }
gfCNCPoint5[8430] = {X 543.6918, Y 54.6769, Z -7.1667, A 0.000, B 0.000, C 0.000 }
gfCNCPoint5[8431] = {X 526.1845, Y 54.6772, Z -7.1667, A 0.000, B 0.000, C 0.000 }
gfCNCPoint5[8432] = {X 524.8901, Y 55.4738, Z -7.1667, A 0.000, B 0.000, C 0.000 }
gfCNCPoint5[8433] = {X 523.4884, Y 56.0614, Z -7.1667, A 0.000, B 0.000, C 0.000 }
gfCNCPoint5[8434] = {X 522.0130, Y 56.4261, Z -7.1667, A 0.000, B 0.000, C 0.000 }
gfCNCPoint5[8435] = {X 520.4990, Y 56.5591, Z -7.1667, A 0.000, B 0.000, C 0.000 }
gfCNCPoint5[8436] = {X 519.7998, Y 56.5591, Z -7.1667, A 0.000, B 0.000, C 0.000 }
gfCNCPoint5[8437] = {X 518.3493, Y 56.4498, Z -7.1667, A 0.000, B 0.000, C 0.000 }
gfCNCPoint5[8438] = {X 516.9316, Y 56.1244, Z -7.1667, A 0.000, B 0.000, C 0.000 }
gfCNCPoint5[8439] = {X 515.5787, Y 55.5903, Z -7.1667, A 0.000, B 0.000, C 0.000 }
gfCNCPoint5[8440] = {X 514.3210, Y 54.8595, Z -7.1667, A 0.000, B 0.000, C 0.000 }
gfCNCPoint5[8441] = {X 513.1871, Y 53.9484, Z -7.1667, A 0.000, B 0.000, C 0.000 }
gfCNCPoint5[8442] = {X 512.2025, Y 52.8778, Z -7.1667, A 0.000, B 0.000, C 0.000 }
gfCNCPoint5[8443] = {X 511.3855, Y 51.6648, Z -7.1667, A 0.000, B 0.000, C 0.000 }
gfCNCPoint5[8444] = {X 510.7606, Y 50.3426, Z -7.1667, A 0.000, B 0.000, C 0.000 }
gfCNCPoint5[8445] = {X 509.8636, Y 51.4977, Z -7.1667, A 0.000, B 0.000, C 0.000 }
gfCNCPoint5[8446] = {X 508.8029, Y 52.5044, Z -7.1667, A 0.000, B 0.000, C 0.000 }
gfCNCPoint5[8447] = {X 507.7229, Y 53.2678, Z -7.1667, A 0.000, B 0.000, C 0.000 }
gfCNCPoint5[8448] = {X 506.5489, Y 53.8769, Z -7.1667, A 0.000, B 0.000, C 0.000 }
gfCNCPoint5[8449] = {X 505.3028, Y 54.3203, Z -7.1667, A 0.000, B 0.000, C 0.000 }
gfCNCPoint5[8450] = {X 504.0080, Y 54.5896, Z -7.1667, A 0.000, B 0.000, C 0.000 }
gfCNCPoint5[8451] = {X 502.6885, Y 54.6800, Z -7.1667, A 0.000, B 0.000, C 0.000 }
gfCNCPoint5[8452] = {X 496.2450, Y 54.6800, Z -7.1667, A 0.000, B 0.000, C 0.000 }
gfCNCPoint5[8453] = {X 495.0285, Y 54.6033, Z -7.1667, A 0.000, B 0.000, C 0.000 }
gfCNCPoint5[8454] = {X 493.8313, Y 54.3742, Z -7.1667, A 0.000, B 0.000, C 0.000 }
gfCNCPoint5[8455] = {X 492.6724, Y 53.9966, Z -7.1667, A 0.000, B 0.000, C 0.000 }
gfCNCPoint5[8456] = {X 491.4451, Y 53.4062, Z -7.1667, A 0.000, B 0.000, C 0.000 }
gfCNCPoint5[8457] = {X 490.3129, Y 52.6493, Z -7.1667, A 0.000, B 0.000, C 0.000 }
gfCNCPoint5[8458] = {X 489.2980, Y 51.7410, Z -7.1667, A 0.000, B 0.000, C 0.000 }
gfCNCPoint5[8459] = {X 488.8683, Y 52.1573, Z -7.1667, A 0.000, B 0.000, C 0.000 }
gfCNCPoint5[8460] = {X 488.4137, Y 52.5463, Z -7.1667, A 0.000, B 0.000, C 0.000 }
gfCNCPoint5[8461] = {X 488.8649, Y 53.8245, Z -7.1667, A 0.000, B 0.000, C 0.000 }
gfCNCPoint5[8462] = {X 489.1946, Y 55.1393, Z -7.1667, A 0.000, B 0.000, C 0.000 }
gfCNCPoint5[8463] = {X 489.3999, Y 56.4792, Z -7.1667, A 0.000, B 0.000, C 0.000 }
gfCNCPoint5[8464] = {X 489.4600, Y 57.2386, Z -7.1667, A 0.000, B 0.000, C 0.000 }
